LIN {X 152.500,Y 49.993,Z 45.000,A 180.000,B 0.000,C 180.000} C_DIS
LIN {X 152.500,Y 49.993,Z 52.000,A 180.000,B 0.000,C 180.000} C_DIS
LIN {X 147.273,Y 49.993,Z 52.000,A 180.000,B 0.000,C 180.000} C_DIS
LIN {X 147.273,Y 49.993,Z 57.000,A 180.000,B 0.000,C 180.000} C_DIS
LIN {X 118.528,Y 49.993,Z 57.000,A 180.000,B 0.000,C 180.000} C_DIS
LIN {X 118.528,Y 49.993,Z 62.000,A 180.000,B 0.000,C 180.000} C_DIS
LIN {X 104.744,Y 49.993,Z 62.000,A 180.000,B 0.000,C 180.000} C_DIS
LIN {X 104.744,Y 49.993,Z 63.247,A 180.000,B 0.000,C 180.000} C_DIS
LIN {X 104.720,Y 49.993,Z 63.811,A 180.000,B 0.000,C 180.000} C_DIS
LIN {X 104.656,Y 49.993,Z 64.331,A 180.000,B 0.000,C 180.000} C_DIS
LIN {X 104.555,Y 49.993,Z 64.841,A 180.000,B 0.000,C 180.000} C_DIS
LIN {X 104.417,Y 49.993,Z 65.337,A 180.000,B 0.000,C 180.000} C_DIS
LIN {X 104.239,Y 49.993,Z 65.829,A 180.000,B 0.000,C 180.000} C_DIS
LIN {X 104.023,Y 49.993,Z 66.308,A 180.000,B 0.000,C 180.000} C_DIS
LIN {X 103.772,Y 49.993,Z 66.769,A 180.000,B 0.000,C 180.000} C_DIS
LIN {X 103.485,Y 49.993,Z 67.212,A 180.000,B 0.000,C 180.000} C_DIS
LIN {X 103.167,Y 49.993,Z 67.630,A 180.000,B 0.000,C 180.000} C_DIS
LIN {X 102.799,Y 49.993,Z 68.043,A 180.000,B 0.000,C 180.000} C_DIS
LIN {X 102.416,Y 49.993,Z 68.409,A 180.000,B 0.000,C 180.000} C_DIS
LIN {X 102.020,Y 49.993,Z 68.735,A 180.000,B 0.000,C 180.000} C_DIS
LIN {X 101.582,Y 49.993,Z 69.044,A 180.000,B 0.000,C 180.000} C_DIS
LIN {X 101.120,Y 49.993,Z 69.322,A 180.000,B 0.000,C 180.000} C_DIS
LIN {X 100.633,Y 49.993,Z 69.567,A 180.000,B 0.000,C 180.000} C_DIS
LIN {X 100.135,Y 49.993,Z 69.771,A 180.000,B 0.000,C 180.000} C_DIS
LIN {X 99.619,Y 49.993,Z 69.940,A 180.000,B 0.000,C 180.000} C_DIS
LIN {X 99.066,Y 49.993,Z 70.078,A 180.000,B 0.000,C 180.000} C_DIS
LIN {X 98.519,Y 49.993,Z 70.171,A 180.000,B 0.000,C 180.000} C_DIS
LIN {X 97.977,Y 49.993,Z 70.227,A 180.000,B 0.000,C 180.000} C_DIS
LIN {X 97.314,Y 49.993,Z 70.247,A 180.000,B 0.000,C 180.000} C_DIS
LIN {X 95.979,Y 49.993,Z 70.247,A 180.000,B 0.000,C 180.000} C_DIS
LIN {X 95.978,Y 49.993,Z 72.155,A 180.000,B 0.000,C 180.000} C_DIS
LIN {X 90.667,Y 49.993,Z 74.364,A 180.000,B 0.000,C 180.000} C_DIS
LIN {X 85.391,Y 49.993,Z 74.361,A 180.000,B 0.000,C 180.000} C_DIS
LIN {X 84.621,Y 49.993,Z 73.716,A 180.000,B 0.000,C 180.000} C_DIS
LIN {X 83.893,Y 49.993,Z 73.150,A 180.000,B 0.000,C 180.000} C_DIS
LIN {X 83.135,Y 49.993,Z 72.607,A 180.000,B 0.000,C 180.000} C_DIS
LIN {X 82.449,Y 49.993,Z 72.157,A 180.000,B 0.000,C 180.000} C_DIS
LIN {X 81.782,Y 49.993,Z 71.760,A 180.000,B 0.000,C 180.000} C_DIS
LIN {X 81.128,Y 49.993,Z 71.411,A 180.000,B 0.000,C 180.000} C_DIS
LIN {X 80.479,Y 49.993,Z 71.101,A 180.000,B 0.000,C 180.000} C_DIS
LIN {X 79.861,Y 49.993,Z 70.843,A 180.000,B 0.000,C 180.000} C_DIS
LIN {X 79.251,Y 49.993,Z 70.625,A 180.000,B 0.000,C 180.000} C_DIS
LIN {X 78.642,Y 49.993,Z 70.441,A 180.000,B 0.000,C 180.000} C_DIS
LIN {X 78.537,Y 49.993,Z 70.415,A 180.000,B 0.000,C 180.000} C_DIS
LIN {X 78.116,Y 49.993,Z 70.531,A 180.000,B 0.000,C 180.000} C_DIS
LIN {X 77.493,Y 49.993,Z 70.735,A 180.000,B 0.000,C 180.000} C_DIS
LIN {X 76.864,Y 49.993,Z 70.978,A 180.000,B 0.000,C 180.000} C_DIS
LIN {X 76.232,Y 49.993,Z 71.257,A 180.000,B 0.000,C 180.000} C_DIS
LIN {X 75.610,Y 49.993,Z 71.566,A 180.000,B 0.000,C 180.000} C_DIS
LIN {X 74.985,Y 49.993,Z 71.907,A 180.000,B 0.000,C 180.000} C_DIS
LIN {X 74.357,Y 49.993,Z 72.279,A 180.000,B 0.000,C 180.000} C_DIS
LIN {X 73.718,Y 49.993,Z 72.687,A 180.000,B 0.000,C 180.000} C_DIS
LIN {X 73.038,Y 49.993,Z 73.149,A 180.000,B 0.000,C 180.000} C_DIS
LIN {X 72.140,Y 49.993,Z 73.798,A 180.000,B 0.000,C 180.000} C_DIS
LIN {X 71.311,Y 49.993,Z 74.436,A 180.000,B 0.000,C 180.000} C_DIS
LIN {X 70.169,Y 49.993,Z 75.345,A 180.000,B 0.000,C 180.000} C_DIS
LIN {X 66.951,Y 49.993,Z 77.983,A 180.000,B 0.000,C 180.000} C_DIS
LIN {X 65.792,Y 49.993,Z 78.895,A 180.000,B 0.000,C 180.000} C_DIS
LIN {X 65.177,Y 49.993,Z 79.359,A 180.000,B 0.000,C 180.000} C_DIS
LIN {X 64.612,Y 49.993,Z 79.770,A 180.000,B 0.000,C 180.000} C_DIS
LIN {X 64.036,Y 49.993,Z 80.171,A 180.000,B 0.000,C 180.000} C_DIS
LIN {X 63.450,Y 49.993,Z 80.559,A 180.000,B 0.000,C 180.000} C_DIS
LIN {X 62.857,Y 49.993,Z 80.929,A 180.000,B 0.000,C 180.000} C_DIS
LIN {X 62.256,Y 49.993,Z 81.279,A 180.000,B 0.000,C 180.000} C_DIS
LIN {X 61.642,Y 49.993,Z 81.610,A 180.000,B 0.000,C 180.000} C_DIS
LIN {X 61.028,Y 49.993,Z 81.911,A 180.000,B 0.000,C 180.000} C_DIS
LIN {X 60.400,Y 49.993,Z 82.187,A 180.000,B 0.000,C 180.000} C_DIS
LIN {X 59.765,Y 49.993,Z 82.432,A 180.000,B 0.000,C 180.000} C_DIS
LIN {X 59.120,Y 49.993,Z 82.646,A 180.000,B 0.000,C 180.000} C_DIS
LIN {X 58.464,Y 49.993,Z 82.825,A 180.000,B 0.000,C 180.000} C_DIS
LIN {X 57.793,Y 49.993,Z 82.968,A 180.000,B 0.000,C 180.000} C_DIS
LIN {X 57.412,Y 49.993,Z 83.031,A 180.000,B 0.000,C 180.000} C_DIS
LIN {X 57.076,Y 49.993,Z 83.075,A 180.000,B 0.000,C 180.000} C_DIS
LIN {X 56.731,Y 49.993,Z 83.110,A 180.000,B 0.000,C 180.000} C_DIS
LIN {X 56.398,Y 49.993,Z 83.133,A 180.000,B 0.000,C 180.000} C_DIS
LIN {X 56.071,Y 49.993,Z 83.146,A 180.000,B 0.000,C 180.000} C_DIS
LIN {X 55.283,Y 49.993,Z 83.150,A 180.000,B 0.000,C 180.000} C_DIS
LIN {X 50.550,Y 49.993,Z 83.146,A 180.000,B 0.000,C 180.000} C_DIS
LIN {X 50.101,Y 49.993,Z 83.124,A 180.000,B 0.000,C 180.000} C_DIS
LIN {X 49.670,Y 49.993,Z 83.075,A 180.000,B 0.000,C 180.000} C_DIS
LIN {X 49.319,Y 49.993,Z 83.017,A 180.000,B 0.000,C 180.000} C_DIS
LIN {X 48.906,Y 49.993,Z 82.926,A 180.000,B 0.000,C 180.000} C_DIS
LIN {X 48.508,Y 49.993,Z 82.808,A 180.000,B 0.000,C 180.000} C_DIS
LIN {X 48.202,Y 49.993,Z 82.700,A 180.000,B 0.000,C 180.000} C_DIS
LIN {X 47.898,Y 49.993,Z 82.574,A 180.000,B 0.000,C 180.000} C_DIS
LIN {X 47.607,Y 49.993,Z 82.435,A 180.000,B 0.000,C 180.000} C_DIS
LIN {X 47.311,Y 49.993,Z 82.272,A 180.000,B 0.000,C 180.000} C_DIS
LIN {X 46.970,Y 49.993,Z 82.051,A 180.000,B 0.000,C 180.000} C_DIS
LIN {X 46.686,Y 49.993,Z 81.832,A 180.000,B 0.000,C 180.000} C_DIS
LIN {X 46.466,Y 49.993,Z 81.631,A 180.000,B 0.000,C 180.000} C_DIS
LIN {X 46.280,Y 49.993,Z 81.428,A 180.000,B 0.000,C 180.000} C_DIS
LIN {X 46.138,Y 49.993,Z 81.234,A 180.000,B 0.000,C 180.000} C_DIS
LIN {X 46.052,Y 49.993,Z 81.067,A 180.000,B 0.000,C 180.000} C_DIS
LIN {X 46.015,Y 49.993,Z 80.948,A 180.000,B 0.000,C 180.000} C_DIS
LIN {X 46.006,Y 49.993,Z 80.865,A 180.000,B 0.000,C 180.000} C_DIS
LIN {X 46.006,Y 49.993,Z 62.000,A 180.000,B 0.000,C 180.000} C_DIS
LIN {X 36.472,Y 49.993,Z 62.000,A 180.000,B 0.000,C 180.000} C_DIS
LIN {X 36.472,Y 49.993,Z 57.000,A 180.000,B 0.000,C 180.000} C_DIS
LIN {X 7.727,Y 49.993,Z 57.000,A 180.000,B 0.000,C 180.000} C_DIS
LIN {X 7.727,Y 49.993,Z 52.000,A 180.000,B 0.000,C 180.000} C_DIS
LIN {X 2.500,Y 49.993,Z 52.000,A 180.000,B 0.000,C 180.000} C_DIS
LIN {X 2.500,Y 49.993,Z 45.000,A 180.000,B 0.000,C 180.000} C_DIS
LIN {X -0.010,Y 49.993,Z 45.000,A 180.000,B 0.000,C 180.000} C_DIS
; Link Move Starts
LIN {X -0.120,Y 49.993,Z 45.026,A 180.000,B 0.000,C 180.000} C_DIS
LIN {X -0.230,Y 49.993,Z 45.051,A 180.000,B 0.000,C 180.000} C_DIS
LIN {X -0.771,Y 50.305,Z 45.051,A 180.000,B 0.000,C 180.000} C_DIS
LIN {X -0.771,Y 50.930,Z 45.051,A 180.000,B 0.000,C 180.000} C_DIS
LIN {X -0.230,Y 51.243,Z 45.051,A 180.000,B 0.000,C 180.000} C_DIS
LIN {X -0.120,Y 51.243,Z 45.026,A 180.000,B 0.000,C 180.000} C_DIS
LIN {X -0.010,Y 51.243,Z 45.000,A 180.000,B 0.000,C 180.000} C_DIS
; Cutting Move Starts
LIN {X 2.500,Y 51.243,Z 45.000,A 180.000,B 0.000,C 180.000} C_DIS
LIN {X 2.500,Y 51.243,Z 52.000,A 180.000,B 0.000,C 180.000} C_DIS
LIN {X 7.251,Y 51.243,Z 52.000,A 180.000,B 0.000,C 180.000} C_DIS
LIN {X 7.251,Y 51.243,Z 57.000,A 180.000,B 0.000,C 180.000} C_DIS
LIN {X 35.222,Y 51.243,Z 57.000,A 180.000,B 0.000,C 180.000} C_DIS
LIN {X 35.222,Y 51.243,Z 62.000,A 180.000,B 0.000,C 180.000} C_DIS
LIN {X 44.115,Y 51.243,Z 62.000,A 180.000,B 0.000,C 180.000} C_DIS
LIN {X 44.117,Y 51.243,Z 80.467,A 180.000,B 0.000,C 180.000} C_DIS
LIN {X 44.271,Y 51.243,Z 80.606,A 180.000,B 0.000,C 180.000} C_DIS
LIN {X 44.597,Y 51.243,Z 80.888,A 180.000,B 0.000,C 180.000} C_DIS
LIN {X 44.947,Y 51.243,Z 81.164,A 180.000,B 0.000,C 180.000} C_DIS
LIN {X 45.375,Y 51.243,Z 81.471,A 180.000,B 0.000,C 180.000} C_DIS
LIN {X 45.822,Y 51.243,Z 81.755,A 180.000,B 0.000,C 180.000} C_DIS
LIN {X 46.192,Y 51.243,Z 81.966,A 180.000,B 0.000,C 180.000} C_DIS
LIN {X 46.558,Y 51.243,Z 82.155,A 180.000,B 0.000,C 180.000} C_DIS
LIN {X 46.947,Y 51.243,Z 82.336,A 180.000,B 0.000,C 180.000} C_DIS
LIN {X 47.425,Y 51.243,Z 82.530,A 180.000,B 0.000,C 180.000} C_DIS
LIN {X 47.877,Y 51.243,Z 82.685,A 180.000,B 0.000,C 180.000} C_DIS
LIN {X 48.271,Y 51.243,Z 82.801,A 180.000,B 0.000,C 180.000} C_DIS
LIN {X 48.688,Y 51.243,Z 82.904,A 180.000,B 0.000,C 180.000} C_DIS
LIN {X 49.230,Y 51.243,Z 83.010,A 180.000,B 0.000,C 180.000} C_DIS
LIN {X 49.667,Y 51.243,Z 83.072,A 180.000,B 0.000,C 180.000} C_DIS
LIN {X 50.108,Y 51.243,Z 83.116,A 180.000,B 0.000,C 180.000} C_DIS
LIN {X 50.473,Y 51.243,Z 83.138,A 180.000,B 0.000,C 180.000} C_DIS
LIN {X 50.806,Y 51.243,Z 83.148,A 180.000,B 0.000,C 180.000} C_DIS
LIN {X 55.704,Y 51.243,Z 83.150,A 180.000,B 0.000,C 180.000} C_DIS
LIN {X 56.493,Y 51.243,Z 83.146,A 180.000,B 0.000,C 180.000} C_DIS
LIN {X 56.819,Y 51.243,Z 83.133,A 180.000,B 0.000,C 180.000} C_DIS
LIN {X 57.153,Y 51.243,Z 83.110,A 180.000,B 0.000,C 180.000} C_DIS
LIN {X 57.497,Y 51.243,Z 83.075,A 180.000,B 0.000,C 180.000} C_DIS
LIN {X 57.833,Y 51.243,Z 83.031,A 180.000,B 0.000,C 180.000} C_DIS
LIN {X 58.213,Y 51.243,Z 82.968,A 180.000,B 0.000,C 180.000} C_DIS
LIN {X 58.886,Y 51.243,Z 82.825,A 180.000,B 0.000,C 180.000} C_DIS
LIN {X 59.541,Y 51.243,Z 82.646,A 180.000,B 0.000,C 180.000} C_DIS
LIN {X 60.187,Y 51.243,Z 82.432,A 180.000,B 0.000,C 180.000} C_DIS
LIN {X 60.822,Y 51.243,Z 82.187,A 180.000,B 0.000,C 180.000} C_DIS
LIN {X 61.450,Y 51.243,Z 81.911,A 180.000,B 0.000,C 180.000} C_DIS
LIN {X 62.064,Y 51.243,Z 81.610,A 180.000,B 0.000,C 180.000} C_DIS
LIN {X 62.677,Y 51.243,Z 81.279,A 180.000,B 0.000,C 180.000} C_DIS
LIN {X 63.279,Y 51.243,Z 80.929,A 180.000,B 0.000,C 180.000} C_DIS
LIN {X 63.872,Y 51.243,Z 80.559,A 180.000,B 0.000,C 180.000} C_DIS
LIN {X 64.458,Y 51.243,Z 80.171,A 180.000,B 0.000,C 180.000} C_DIS
LIN {X 65.033,Y 51.243,Z 79.770,A 180.000,B 0.000,C 180.000} C_DIS
LIN {X 65.598,Y 51.243,Z 79.359,A 180.000,B 0.000,C 180.000} C_DIS
LIN {X 66.214,Y 51.243,Z 78.896,A 180.000,B 0.000,C 180.000} C_DIS
LIN {X 67.373,Y 51.243,Z 77.983,A 180.000,B 0.000,C 180.000} C_DIS
LIN {X 70.591,Y 51.243,Z 75.345,A 180.000,B 0.000,C 180.000} C_DIS
LIN {X 71.733,Y 51.243,Z 74.436,A 180.000,B 0.000,C 180.000} C_DIS
LIN {X 72.562,Y 51.243,Z 73.798,A 180.000,B 0.000,C 180.000} C_DIS
LIN {X 73.460,Y 51.243,Z 73.149,A 180.000,B 0.000,C 180.000} C_DIS
LIN {X 74.139,Y 51.243,Z 72.687,A 180.000,B 0.000,C 180.000} C_DIS
LIN {X 74.779,Y 51.243,Z 72.279,A 180.000,B 0.000,C 180.000} C_DIS
LIN {X 75.406,Y 51.243,Z 71.907,A 180.000,B 0.000,C 180.000} C_DIS
LIN {X 76.031,Y 51.243,Z 71.566,A 180.000,B 0.000,C 180.000} C_DIS
LIN {X 76.653,Y 51.243,Z 71.257,A 180.000,B 0.000,C 180.000} C_DIS
LIN {X 77.286,Y 51.243,Z 70.978,A 180.000,B 0.000,C 180.000} C_DIS
LIN {X 77.914,Y 51.243,Z 70.735,A 180.000,B 0.000,C 180.000} C_DIS
LIN {X 78.537,Y 51.243,Z 70.531,A 180.000,B 0.000,C 180.000} C_DIS
LIN {X 78.959,Y 51.243,Z 70.415,A 180.000,B 0.000,C 180.000} C_DIS
LIN {X 79.064,Y 51.243,Z 70.441,A 180.000,B 0.000,C 180.000} C_DIS
LIN {X 79.672,Y 51.243,Z 70.625,A 180.000,B 0.000,C 180.000} C_DIS
LIN {X 80.283,Y 51.243,Z 70.843,A 180.000,B 0.000,C 180.000} C_DIS
LIN {X 80.901,Y 51.243,Z 71.101,A 180.000,B 0.000,C 180.000} C_DIS
LIN {X 81.550,Y 51.243,Z 71.411,A 180.000,B 0.000,C 180.000} C_DIS
LIN {X 82.204,Y 51.243,Z 71.760,A 180.000,B 0.000,C 180.000} C_DIS
LIN {X 82.871,Y 51.243,Z 72.157,A 180.000,B 0.000,C 180.000} C_DIS
LIN {X 83.557,Y 51.243,Z 72.607,A 180.000,B 0.000,C 180.000} C_DIS
LIN {X 84.314,Y 51.243,Z 73.150,A 180.000,B 0.000,C 180.000} C_DIS
LIN {X 85.043,Y 51.243,Z 73.716,A 180.000,B 0.000,C 180.000} C_DIS
LIN {X 85.812,Y 51.243,Z 74.361,A 180.000,B 0.000,C 180.000} C_DIS
LIN {X 91.091,Y 51.243,Z 74.364,A 180.000,B 0.000,C 180.000} C_DIS
LIN {X 96.400,Y 51.243,Z 72.155,A 180.000,B 0.000,C 180.000} C_DIS
LIN {X 96.401,Y 51.243,Z 70.247,A 180.000,B 0.000,C 180.000} C_DIS
LIN {X 96.436,Y 51.243,Z 70.247,A 180.000,B 0.000,C 180.000} C_DIS
LIN {X 97.201,Y 51.243,Z 70.228,A 180.000,B 0.000,C 180.000} C_DIS
LIN {X 97.835,Y 51.243,Z 70.171,A 180.000,B 0.000,C 180.000} C_DIS
LIN {X 98.445,Y 51.243,Z 70.077,A 180.000,B 0.000,C 180.000} C_DIS
LIN {X 99.048,Y 51.243,Z 69.941,A 180.000,B 0.000,C 180.000} C_DIS
LIN {X 99.604,Y 51.243,Z 69.772,A 180.000,B 0.000,C 180.000} C_DIS
LIN {X 100.142,Y 51.243,Z 69.564,A 180.000,B 0.000,C 180.000} C_DIS
LIN {X 100.650,Y 51.243,Z 69.326,A 180.000,B 0.000,C 180.000} C_DIS
LIN {X 101.144,Y 51.243,Z 69.043,A 180.000,B 0.000,C 180.000} C_DIS
LIN {X 101.601,Y 51.243,Z 68.735,A 180.000,B 0.000,C 180.000} C_DIS
LIN {X 102.028,Y 51.243,Z 68.398,A 180.000,B 0.000,C 180.000} C_DIS
LIN {X 102.427,Y 51.243,Z 68.030,A 180.000,B 0.000,C 180.000} C_DIS
LIN {X 102.794,Y 51.243,Z 67.630,A 180.000,B 0.000,C 180.000} C_DIS
LIN {X 103.123,Y 51.243,Z 67.212,A 180.000,B 0.000,C 180.000} C_DIS
LIN {X 103.421,Y 51.243,Z 66.768,A 180.000,B 0.000,C 180.000} C_DIS
LIN {X 103.681,Y 51.243,Z 66.307,A 180.000,B 0.000,C 180.000} C_DIS
LIN {X 103.905,Y 51.243,Z 65.828,A 180.000,B 0.000,C 180.000} C_DIS
LIN {X 104.090,Y 51.243,Z 65.333,A 180.000,B 0.000,C 180.000} C_DIS
LIN {X 104.228,Y 51.243,Z 64.853,A 180.000,B 0.000,C 180.000} C_DIS
LIN {X 104.335,Y 51.243,Z 64.336,A 180.000,B 0.000,C 180.000} C_DIS
LIN {X 104.400,Y 51.243,Z 63.822,A 180.000,B 0.000,C 180.000} C_DIS
LIN {X 104.422,Y 51.243,Z 63.353,A 180.000,B 0.000,C 180.000} C_DIS
LIN {X 104.427,Y 51.243,Z 62.000,A 180.000,B 0.000,C 180.000} C_DIS
LIN {X 119.778,Y 51.243,Z 62.000,A 180.000,B 0.000,C 180.000} C_DIS
LIN {X 119.778,Y 51.243,Z 57.000,A 180.000,B 0.000,C 180.000} C_DIS
LIN {X 147.749,Y 51.243,Z 57.000,A 180.000,B 0.000,C 180.000} C_DIS
LIN {X 147.749,Y 51.243,Z 52.000,A 180.000,B 0.000,C 180.000} C_DIS
LIN {X 152.500,Y 51.243,Z 52.000,A 180.000,B 0.000,C 180.000} C_DIS
LIN {X 152.500,Y 51.243,Z 45.000,A 180.000,B 0.000,C 180.000} C_DIS
LIN {X 155.010,Y 51.243,Z 45.000,A 180.000,B 0.000,C 180.000} C_DIS
; Link Move Starts
LIN {X 155.120,Y 51.243,Z 45.026,A 180.000,B 0.000,C 180.000} C_DIS
LIN {X 155.230,Y 51.243,Z 45.051,A 180.000,B 0.000,C 180.000} C_DIS
LIN {X 155.771,Y 51.555,Z 45.051,A 180.000,B 0.000,C 180.000} C_DIS
LIN {X 155.771,Y 52.180,Z 45.051,A 180.000,B 0.000,C 180.000} C_DIS
LIN {X 155.230,Y 52.492,Z 45.051,A 180.000,B 0.000,C 180.000} C_DIS
LIN {X 155.120,Y 52.492,Z 45.026,A 180.000,B 0.000,C 180.000} C_DIS
LIN {X 155.010,Y 52.492,Z 45.000,A 180.000,B 0.000,C 180.000} C_DIS
; Cutting Move Starts
LIN {X 152.500,Y 52.492,Z 45.000,A 180.000,B 0.000,C 180.000} C_DIS
LIN {X 152.500,Y 52.492,Z 52.000,A 180.000,B 0.000,C 180.000} C_DIS
LIN {X 148.203,Y 52.492,Z 52.000,A 180.000,B 0.000,C 180.000} C_DIS
LIN {X 148.199,Y 52.492,Z 57.000,A 180.000,B 0.000,C 180.000} C_DIS
LIN {X 121.028,Y 52.492,Z 57.000,A 180.000,B 0.000,C 180.000} C_DIS
LIN {X 121.028,Y 52.492,Z 62.000,A 180.000,B 0.000,C 180.000} C_DIS
LIN {X 103.956,Y 52.492,Z 62.000,A 180.000,B 0.000,C 180.000} C_DIS
LIN {X 103.953,Y 52.492,Z 63.301,A 180.000,B 0.000,C 180.000} C_DIS
LIN {X 103.931,Y 52.492,Z 63.800,A 180.000,B 0.000,C 180.000} C_DIS
LIN {X 103.865,Y 52.492,Z 64.320,A 180.000,B 0.000,C 180.000} C_DIS
LIN {X 103.757,Y 52.492,Z 64.831,A 180.000,B 0.000,C 180.000} C_DIS
LIN {X 103.610,Y 52.492,Z 65.333,A 180.000,B 0.000,C 180.000} C_DIS
LIN {X 103.411,Y 52.492,Z 65.843,A 180.000,B 0.000,C 180.000} C_DIS
LIN {X 103.185,Y 52.492,Z 66.305,A 180.000,B 0.000,C 180.000} C_DIS
LIN {X 102.912,Y 52.492,Z 66.765,A 180.000,B 0.000,C 180.000} C_DIS
LIN {X 102.599,Y 52.492,Z 67.209,A 180.000,B 0.000,C 180.000} C_DIS
LIN {X 102.251,Y 52.492,Z 67.628,A 180.000,B 0.000,C 180.000} C_DIS
LIN {X 101.862,Y 52.492,Z 68.029,A 180.000,B 0.000,C 180.000} C_DIS
LIN {X 101.440,Y 52.492,Z 68.395,A 180.000,B 0.000,C 180.000} C_DIS
LIN {X 100.981,Y 52.492,Z 68.734,A 180.000,B 0.000,C 180.000} C_DIS
LIN {X 100.490,Y 52.492,Z 69.044,A 180.000,B 0.000,C 180.000} C_DIS
LIN {X 99.962,Y 52.492,Z 69.319,A 180.000,B 0.000,C 180.000} C_DIS
LIN {X 99.400,Y 52.492,Z 69.562,A 180.000,B 0.000,C 180.000} C_DIS
LIN {X 98.791,Y 52.492,Z 69.772,A 180.000,B 0.000,C 180.000} C_DIS
LIN {X 98.157,Y 52.492,Z 69.940,A 180.000,B 0.000,C 180.000} C_DIS
LIN {X 97.461,Y 52.492,Z 70.075,A 180.000,B 0.000,C 180.000} C_DIS
LIN {X 96.823,Y 52.492,Z 70.157,A 180.000,B 0.000,C 180.000} C_DIS
LIN {X 96.820,Y 52.492,Z 72.156,A 180.000,B 0.000,C 180.000} C_DIS
LIN {X 91.513,Y 52.492,Z 74.364,A 180.000,B 0.000,C 180.000} C_DIS
LIN {X 86.234,Y 52.492,Z 74.361,A 180.000,B 0.000,C 180.000} C_DIS
LIN {X 85.465,Y 52.492,Z 73.716,A 180.000,B 0.000,C 180.000} C_DIS
LIN {X 84.737,Y 52.492,Z 73.150,A 180.000,B 0.000,C 180.000} C_DIS
LIN {X 83.979,Y 52.492,Z 72.607,A 180.000,B 0.000,C 180.000} C_DIS
LIN {X 83.293,Y 52.492,Z 72.157,A 180.000,B 0.000,C 180.000} C_DIS
LIN {X 82.626,Y 52.492,Z 71.761,A 180.000,B 0.000,C 180.000} C_DIS
LIN {X 81.972,Y 52.492,Z 71.411,A 180.000,B 0.000,C 180.000} C_DIS
LIN {X 81.323,Y 52.492,Z 71.101,A 180.000,B 0.000,C 180.000} C_DIS
LIN {X 80.705,Y 52.492,Z 70.843,A 180.000,B 0.000,C 180.000} C_DIS
LIN {X 80.085,Y 52.492,Z 70.622,A 180.000,B 0.000,C 180.000} C_DIS
LIN {X 79.463,Y 52.492,Z 70.435,A 180.000,B 0.000,C 180.000} C_DIS
LIN {X 79.381,Y 52.492,Z 70.415,A 180.000,B 0.000,C 180.000} C_DIS
LIN {X 78.959,Y 52.492,Z 70.531,A 180.000,B 0.000,C 180.000} C_DIS
LIN {X 78.336,Y 52.492,Z 70.735,A 180.000,B 0.000,C 180.000} C_DIS
LIN {X 77.707,Y 52.492,Z 70.978,A 180.000,B 0.000,C 180.000} C_DIS
LIN {X 77.075,Y 52.492,Z 71.257,A 180.000,B 0.000,C 180.000} C_DIS
LIN {X 76.453,Y 52.492,Z 71.566,A 180.000,B 0.000,C 180.000} C_DIS
LIN {X 75.828,Y 52.492,Z 71.907,A 180.000,B 0.000,C 180.000} C_DIS
LIN {X 75.200,Y 52.492,Z 72.279,A 180.000,B 0.000,C 180.000} C_DIS
LIN {X 74.561,Y 52.492,Z 72.687,A 180.000,B 0.000,C 180.000} C_DIS
LIN {X 73.881,Y 52.492,Z 73.149,A 180.000,B 0.000,C 180.000} C_DIS
LIN {X 72.984,Y 52.492,Z 73.798,A 180.000,B 0.000,C 180.000} C_DIS
LIN {X 72.154,Y 52.492,Z 74.436,A 180.000,B 0.000,C 180.000} C_DIS
LIN {X 71.013,Y 52.492,Z 75.345,A 180.000,B 0.000,C 180.000} C_DIS
LIN {X 67.794,Y 52.492,Z 77.983,A 180.000,B 0.000,C 180.000} C_DIS
LIN {X 66.636,Y 52.492,Z 78.896,A 180.000,B 0.000,C 180.000} C_DIS
LIN {X 66.020,Y 52.492,Z 79.359,A 180.000,B 0.000,C 180.000} C_DIS
LIN {X 65.455,Y 52.492,Z 79.770,A 180.000,B 0.000,C 180.000} C_DIS
LIN {X 64.879,Y 52.492,Z 80.171,A 180.000,B 0.000,C 180.000} C_DIS
LIN {X 64.294,Y 52.492,Z 80.559,A 180.000,B 0.000,C 180.000} C_DIS
LIN {X 63.700,Y 52.492,Z 80.929,A 180.000,B 0.000,C 180.000} C_DIS
LIN {X 63.099,Y 52.492,Z 81.279,A 180.000,B 0.000,C 180.000} C_DIS
LIN {X 62.485,Y 52.492,Z 81.610,A 180.000,B 0.000,C 180.000} C_DIS
LIN {X 61.872,Y 52.492,Z 81.911,A 180.000,B 0.000,C 180.000} C_DIS
LIN {X 61.243,Y 52.492,Z 82.187,A 180.000,B 0.000,C 180.000} C_DIS
LIN {X 60.608,Y 52.492,Z 82.432,A 180.000,B 0.000,C 180.000} C_DIS
LIN {X 59.963,Y 52.492,Z 82.646,A 180.000,B 0.000,C 180.000} C_DIS
LIN {X 59.308,Y 52.492,Z 82.825,A 180.000,B 0.000,C 180.000} C_DIS
LIN {X 58.634,Y 52.492,Z 82.968,A 180.000,B 0.000,C 180.000} C_DIS
LIN {X 58.255,Y 52.492,Z 83.031,A 180.000,B 0.000,C 180.000} C_DIS
LIN {X 57.919,Y 52.492,Z 83.075,A 180.000,B 0.000,C 180.000} C_DIS
LIN {X 57.570,Y 52.492,Z 83.110,A 180.000,B 0.000,C 180.000} C_DIS
LIN {X 57.241,Y 52.492,Z 83.133,A 180.000,B 0.000,C 180.000} C_DIS
LIN {X 56.914,Y 52.492,Z 83.146,A 180.000,B 0.000,C 180.000} C_DIS
LIN {X 56.125,Y 52.492,Z 83.150,A 180.000,B 0.000,C 180.000} C_DIS
LIN {X 51.228,Y 52.492,Z 83.148,A 180.000,B 0.000,C 180.000} C_DIS
LIN {X 50.894,Y 52.492,Z 83.138,A 180.000,B 0.000,C 180.000} C_DIS
LIN {X 50.551,Y 52.492,Z 83.118,A 180.000,B 0.000,C 180.000} C_DIS
LIN {X 50.192,Y 52.492,Z 83.085,A 180.000,B 0.000,C 180.000} C_DIS
LIN {X 49.834,Y 52.492,Z 83.040,A 180.000,B 0.000,C 180.000} C_DIS
LIN {X 49.459,Y 52.492,Z 82.981,A 180.000,B 0.000,C 180.000} C_DIS
LIN {X 49.097,Y 52.492,Z 82.912,A 180.000,B 0.000,C 180.000} C_DIS
LIN {X 48.722,Y 52.492,Z 82.827,A 180.000,B 0.000,C 180.000} C_DIS
LIN {X 48.335,Y 52.492,Z 82.727,A 180.000,B 0.000,C 180.000} C_DIS
LIN {X 47.958,Y 52.492,Z 82.617,A 180.000,B 0.000,C 180.000} C_DIS
LIN {X 47.571,Y 52.492,Z 82.491,A 180.000,B 0.000,C 180.000} C_DIS
LIN {X 47.180,Y 52.492,Z 82.351,A 180.000,B 0.000,C 180.000} C_DIS
LIN {X 46.794,Y 52.492,Z 82.199,A 180.000,B 0.000,C 180.000} C_DIS
LIN {X 46.392,Y 52.492,Z 82.028,A 180.000,B 0.000,C 180.000} C_DIS
LIN {X 45.925,Y 52.492,Z 81.809,A 180.000,B 0.000,C 180.000} C_DIS
LIN {X 45.499,Y 52.492,Z 81.589,A 180.000,B 0.000,C 180.000} C_DIS
LIN {X 45.076,Y 52.492,Z 81.351,A 180.000,B 0.000,C 180.000} C_DIS
LIN {X 44.646,Y 52.492,Z 81.088,A 180.000,B 0.000,C 180.000} C_DIS
LIN {X 44.123,Y 52.492,Z 80.738,A 180.000,B 0.000,C 180.000} C_DIS
LIN {X 43.749,Y 52.492,Z 80.467,A 180.000,B 0.000,C 180.000} C_DIS
LIN {X 43.747,Y 52.492,Z 62.000,A 180.000,B 0.000,C 180.000} C_DIS
LIN {X 33.972,Y 52.492,Z 62.000,A 180.000,B 0.000,C 180.000} C_DIS
LIN {X 33.972,Y 52.492,Z 57.000,A 180.000,B 0.000,C 180.000} C_DIS
LIN {X 6.797,Y 52.492,Z 57.000,A 180.000,B 0.000,C 180.000} C_DIS
LIN {X 6.797,Y 52.492,Z 52.000,A 180.000,B 0.000,C 180.000} C_DIS
LIN {X 2.500,Y 52.492,Z 52.000,A 180.000,B 0.000,C 180.000} C_DIS
LIN {X 2.500,Y 52.492,Z 45.000,A 180.000,B 0.000,C 180.000} C_DIS
LIN {X -0.010,Y 52.492,Z 45.000,A 180.000,B 0.000,C 180.000} C_DIS
; Link Move Starts
LIN {X -0.120,Y 52.492,Z 45.026,A 180.000,B 0.000,C 180.000} C_DIS
LIN {X -0.230,Y 52.492,Z 45.051,A 180.000,B 0.000,C 180.000} C_DIS
LIN {X -0.771,Y 52.805,Z 45.051,A 180.000,B 0.000,C 180.000} C_DIS
LIN {X -0.771,Y 53.430,Z 45.051,A 180.000,B 0.000,C 180.000} C_DIS
LIN {X -0.230,Y 53.742,Z 45.051,A 180.000,B 0.000,C 180.000} C_DIS
LIN {X -0.120,Y 53.742,Z 45.026,A 180.000,B 0.000,C 180.000} C_DIS
LIN {X -0.010,Y 53.742,Z 45.000,A 180.000,B 0.000,C 180.000} C_DIS
; Cutting Move Starts
LIN {X 2.500,Y 53.742,Z 45.000,A 180.000,B 0.000,C 180.000} C_DIS
LIN {X 2.500,Y 53.742,Z 52.000,A 180.000,B 0.000,C 180.000} C_DIS
LIN {X 6.366,Y 53.742,Z 52.000,A 180.000,B 0.000,C 180.000} C_DIS
LIN {X 6.366,Y 53.742,Z 57.000,A 180.000,B 0.000,C 180.000} C_DIS
LIN {X 32.717,Y 53.742,Z 57.000,A 180.000,B 0.000,C 180.000} C_DIS
LIN {X 32.722,Y 53.742,Z 62.000,A 180.000,B 0.000,C 180.000} C_DIS
LIN {X 44.012,Y 53.742,Z 62.000,A 180.000,B 0.000,C 180.000} C_DIS
LIN {X 44.012,Y 53.742,Z 80.467,A 180.000,B 0.000,C 180.000} C_DIS
LIN {X 44.345,Y 53.742,Z 80.684,A 180.000,B 0.000,C 180.000} C_DIS
LIN {X 44.765,Y 53.742,Z 80.947,A 180.000,B 0.000,C 180.000} C_DIS
LIN {X 45.184,Y 53.742,Z 81.196,A 180.000,B 0.000,C 180.000} C_DIS
LIN {X 45.599,Y 53.742,Z 81.428,A 180.000,B 0.000,C 180.000} C_DIS
LIN {X 46.008,Y 53.742,Z 81.643,A 180.000,B 0.000,C 180.000} C_DIS
LIN {X 46.412,Y 53.742,Z 81.843,A 180.000,B 0.000,C 180.000} C_DIS
LIN {X 46.812,Y 53.742,Z 82.027,A 180.000,B 0.000,C 180.000} C_DIS
LIN {X 47.209,Y 53.742,Z 82.196,A 180.000,B 0.000,C 180.000} C_DIS
LIN {X 47.602,Y 53.742,Z 82.351,A 180.000,B 0.000,C 180.000} C_DIS
LIN {X 47.992,Y 53.742,Z 82.491,A 180.000,B 0.000,C 180.000} C_DIS
LIN {X 48.380,Y 53.742,Z 82.617,A 180.000,B 0.000,C 180.000} C_DIS
LIN {X 48.757,Y 53.742,Z 82.727,A 180.000,B 0.000,C 180.000} C_DIS
LIN {X 49.144,Y 53.742,Z 82.827,A 180.000,B 0.000,C 180.000} C_DIS
LIN {X 49.519,Y 53.742,Z 82.912,A 180.000,B 0.000,C 180.000} C_DIS
LIN {X 49.880,Y 53.742,Z 82.981,A 180.000,B 0.000,C 180.000} C_DIS
LIN {X 50.256,Y 53.742,Z 83.040,A 180.000,B 0.000,C 180.000} C_DIS
LIN {X 50.613,Y 53.742,Z 83.085,A 180.000,B 0.000,C 180.000} C_DIS
LIN {X 50.969,Y 53.742,Z 83.117,A 180.000,B 0.000,C 180.000} C_DIS
LIN {X 51.316,Y 53.742,Z 83.138,A 180.000,B 0.000,C 180.000} C_DIS
LIN {X 51.650,Y 53.742,Z 83.148,A 180.000,B 0.000,C 180.000} C_DIS
LIN {X 56.547,Y 53.742,Z 83.150,A 180.000,B 0.000,C 180.000} C_DIS
LIN {X 57.336,Y 53.742,Z 83.146,A 180.000,B 0.000,C 180.000} C_DIS
LIN {X 57.663,Y 53.742,Z 83.133,A 180.000,B 0.000,C 180.000} C_DIS
LIN {X 57.992,Y 53.742,Z 83.110,A 180.000,B 0.000,C 180.000} C_DIS
LIN {X 58.341,Y 53.742,Z 83.075,A 180.000,B 0.000,C 180.000} C_DIS
LIN {X 58.677,Y 53.742,Z 83.031,A 180.000,B 0.000,C 180.000} C_DIS
LIN {X 59.056,Y 53.742,Z 82.968,A 180.000,B 0.000,C 180.000} C_DIS
LIN {X 59.729,Y 53.742,Z 82.825,A 180.000,B 0.000,C 180.000} C_DIS
LIN {X 60.385,Y 53.742,Z 82.646,A 180.000,B 0.000,C 180.000} C_DIS
LIN {X 61.030,Y 53.742,Z 82.432,A 180.000,B 0.000,C 180.000} C_DIS
LIN {X 61.665,Y 53.742,Z 82.187,A 180.000,B 0.000,C 180.000} C_DIS
LIN {X 62.293,Y 53.742,Z 81.911,A 180.000,B 0.000,C 180.000} C_DIS
LIN {X 62.907,Y 53.742,Z 81.610,A 180.000,B 0.000,C 180.000} C_DIS
LIN {X 63.521,Y 53.742,Z 81.279,A 180.000,B 0.000,C 180.000} C_DIS
LIN {X 64.122,Y 53.742,Z 80.929,A 180.000,B 0.000,C 180.000} C_DIS
LIN {X 64.715,Y 53.742,Z 80.559,A 180.000,B 0.000,C 180.000} C_DIS
LIN {X 65.301,Y 53.742,Z 80.171,A 180.000,B 0.000,C 180.000} C_DIS
LIN {X 65.877,Y 53.742,Z 79.770,A 180.000,B 0.000,C 180.000} C_DIS
LIN {X 66.442,Y 53.742,Z 79.359,A 180.000,B 0.000,C 180.000} C_DIS
LIN {X 67.057,Y 53.742,Z 78.895,A 180.000,B 0.000,C 180.000} C_DIS
LIN {X 68.216,Y 53.742,Z 77.983,A 180.000,B 0.000,C 180.000} C_DIS
LIN {X 71.434,Y 53.742,Z 75.345,A 180.000,B 0.000,C 180.000} C_DIS
LIN {X 72.576,Y 53.742,Z 74.436,A 180.000,B 0.000,C 180.000} C_DIS
LIN {X 73.405,Y 53.742,Z 73.798,A 180.000,B 0.000,C 180.000} C_DIS
LIN {X 74.303,Y 53.742,Z 73.149,A 180.000,B 0.000,C 180.000} C_DIS
LIN {X 74.983,Y 53.742,Z 72.687,A 180.000,B 0.000,C 180.000} C_DIS
LIN {X 75.622,Y 53.742,Z 72.279,A 180.000,B 0.000,C 180.000} C_DIS
LIN {X 76.250,Y 53.742,Z 71.907,A 180.000,B 0.000,C 180.000} C_DIS
LIN {X 76.875,Y 53.742,Z 71.566,A 180.000,B 0.000,C 180.000} C_DIS
LIN {X 77.497,Y 53.742,Z 71.257,A 180.000,B 0.000,C 180.000} C_DIS
LIN {X 78.129,Y 53.742,Z 70.978,A 180.000,B 0.000,C 180.000} C_DIS
LIN {X 78.758,Y 53.742,Z 70.735,A 180.000,B 0.000,C 180.000} C_DIS
LIN {X 79.381,Y 53.742,Z 70.531,A 180.000,B 0.000,C 180.000} C_DIS
LIN {X 79.803,Y 53.742,Z 70.415,A 180.000,B 0.000,C 180.000} C_DIS
LIN {X 79.885,Y 53.742,Z 70.435,A 180.000,B 0.000,C 180.000} C_DIS
LIN {X 80.508,Y 53.742,Z 70.622,A 180.000,B 0.000,C 180.000} C_DIS
LIN {X 81.128,Y 53.742,Z 70.844,A 180.000,B 0.000,C 180.000} C_DIS
LIN {X 81.746,Y 53.742,Z 71.102,A 180.000,B 0.000,C 180.000} C_DIS
LIN {X 82.394,Y 53.742,Z 71.411,A 180.000,B 0.000,C 180.000} C_DIS
LIN {X 83.048,Y 53.742,Z 71.761,A 180.000,B 0.000,C 180.000} C_DIS
LIN {X 83.715,Y 53.742,Z 72.158,A 180.000,B 0.000,C 180.000} C_DIS
LIN {X 84.401,Y 53.742,Z 72.608,A 180.000,B 0.000,C 180.000} C_DIS
LIN {X 85.159,Y 53.742,Z 73.150,A 180.000,B 0.000,C 180.000} C_DIS
LIN {X 85.887,Y 53.742,Z 73.717,A 180.000,B 0.000,C 180.000} C_DIS
LIN {X 86.659,Y 53.742,Z 74.364,A 180.000,B 0.000,C 180.000} C_DIS
LIN {X 91.933,Y 53.742,Z 74.364,A 180.000,B 0.000,C 180.000} C_DIS
LIN {X 97.243,Y 53.742,Z 72.156,A 180.000,B 0.000,C 180.000} C_DIS
LIN {X 97.244,Y 53.742,Z 69.838,A 180.000,B 0.000,C 180.000} C_DIS
LIN {X 97.601,Y 53.742,Z 69.760,A 180.000,B 0.000,C 180.000} C_DIS
LIN {X 98.252,Y 53.742,Z 69.574,A 180.000,B 0.000,C 180.000} C_DIS
LIN {X 98.394,Y 53.742,Z 69.527,A 180.000,B 0.000,C 180.000} C_DIS
LIN {X 99.002,Y 53.742,Z 69.299,A 180.000,B 0.000,C 180.000} C_DIS
LIN {X 99.556,Y 53.742,Z 69.043,A 180.000,B 0.000,C 180.000} C_DIS
LIN {X 100.127,Y 53.742,Z 68.725,A 180.000,B 0.000,C 180.000} C_DIS
LIN {X 100.617,Y 53.742,Z 68.393,A 180.000,B 0.000,C 180.000} C_DIS
LIN {X 101.095,Y 53.742,Z 68.014,A 180.000,B 0.000,C 180.000} C_DIS
LIN {X 101.502,Y 53.742,Z 67.630,A 180.000,B 0.000,C 180.000} C_DIS
LIN {X 101.880,Y 53.742,Z 67.207,A 180.000,B 0.000,C 180.000} C_DIS
LIN {X 102.215,Y 53.742,Z 66.764,A 180.000,B 0.000,C 180.000} C_DIS
LIN {X 102.500,Y 53.742,Z 66.319,A 180.000,B 0.000,C 180.000} C_DIS
LIN {X 102.756,Y 53.742,Z 65.823,A 180.000,B 0.000,C 180.000} C_DIS
LIN {X 102.956,Y 53.742,Z 65.333,A 180.000,B 0.000,C 180.000} C_DIS
LIN {X 103.116,Y 53.742,Z 64.822,A 180.000,B 0.000,C 180.000} C_DIS
LIN {X 103.225,Y 53.742,Z 64.328,A 180.000,B 0.000,C 180.000} C_DIS
LIN {X 103.296,Y 53.742,Z 63.810,A 180.000,B 0.000,C 180.000} C_DIS
LIN {X 103.321,Y 53.742,Z 63.314,A 180.000,B 0.000,C 180.000} C_DIS
LIN {X 103.324,Y 53.742,Z 62.000,A 180.000,B 0.000,C 180.000} C_DIS
LIN {X 122.278,Y 53.742,Z 62.000,A 180.000,B 0.000,C 180.000} C_DIS
LIN {X 122.278,Y 53.742,Z 57.000,A 180.000,B 0.000,C 180.000} C_DIS
LIN {X 148.634,Y 53.742,Z 57.000,A 180.000,B 0.000,C 180.000} C_DIS
LIN {X 148.634,Y 53.742,Z 52.000,A 180.000,B 0.000,C 180.000} C_DIS
LIN {X 152.500,Y 53.742,Z 52.000,A 180.000,B 0.000,C 180.000} C_DIS
LIN {X 152.500,Y 53.742,Z 45.000,A 180.000,B 0.000,C 180.000} C_DIS
LIN {X 155.010,Y 53.742,Z 45.000,A 180.000,B 0.000,C 180.000} C_DIS
; Link Move Starts
LIN {X 155.120,Y 53.742,Z 45.026,A 180.000,B 0.000,C 180.000} C_DIS
LIN {X 155.230,Y 53.742,Z 45.051,A 180.000,B 0.000,C 180.000} C_DIS
LIN {X 155.771,Y 54.055,Z 45.051,A 180.000,B 0.000,C 180.000} C_DIS
LIN {X 155.771,Y 54.680,Z 45.051,A 180.000,B 0.000,C 180.000} C_DIS
LIN {X 155.230,Y 54.992,Z 45.051,A 180.000,B 0.000,C 180.000} C_DIS
LIN {X 155.120,Y 54.992,Z 45.026,A 180.000,B 0.000,C 180.000} C_DIS
LIN {X 155.010,Y 54.992,Z 45.000,A 180.000,B 0.000,C 180.000} C_DIS
; Cutting Move Starts
LIN {X 152.500,Y 54.992,Z 45.000,A 180.000,B 0.000,C 180.000} C_DIS
LIN {X 152.500,Y 54.992,Z 52.000,A 180.000,B 0.000,C 180.000} C_DIS
LIN {X 149.043,Y 54.992,Z 52.000,A 180.000,B 0.000,C 180.000} C_DIS
LIN {X 149.041,Y 54.992,Z 57.000,A 180.000,B 0.000,C 180.000} C_DIS
LIN {X 123.528,Y 54.992,Z 57.000,A 180.000,B 0.000,C 180.000} C_DIS
LIN {X 123.528,Y 54.992,Z 62.000,A 180.000,B 0.000,C 180.000} C_DIS
LIN {X 102.500,Y 54.992,Z 62.000,A 180.000,B 0.000,C 180.000} C_DIS
LIN {X 102.497,Y 54.992,Z 63.302,A 180.000,B 0.000,C 180.000} C_DIS
LIN {X 102.470,Y 54.992,Z 63.804,A 180.000,B 0.000,C 180.000} C_DIS
LIN {X 102.393,Y 54.992,Z 64.325,A 180.000,B 0.000,C 180.000} C_DIS
LIN {X 102.268,Y 54.992,Z 64.838,A 180.000,B 0.000,C 180.000} C_DIS
LIN {X 102.103,Y 54.992,Z 65.325,A 180.000,B 0.000,C 180.000} C_DIS
LIN {X 101.881,Y 54.992,Z 65.826,A 180.000,B 0.000,C 180.000} C_DIS
LIN {X 101.614,Y 54.992,Z 66.297,A 180.000,B 0.000,C 180.000} C_DIS
LIN {X 101.288,Y 54.992,Z 66.762,A 180.000,B 0.000,C 180.000} C_DIS
LIN {X 100.916,Y 54.992,Z 67.207,A 180.000,B 0.000,C 180.000} C_DIS
LIN {X 100.518,Y 54.992,Z 67.608,A 180.000,B 0.000,C 180.000} C_DIS
LIN {X 100.015,Y 54.992,Z 68.024,A 180.000,B 0.000,C 180.000} C_DIS
LIN {X 99.581,Y 54.992,Z 68.329,A 180.000,B 0.000,C 180.000} C_DIS
LIN {X 99.466,Y 54.992,Z 68.402,A 180.000,B 0.000,C 180.000} C_DIS
LIN {X 98.889,Y 54.992,Z 68.732,A 180.000,B 0.000,C 180.000} C_DIS
LIN {X 98.217,Y 54.992,Z 69.041,A 180.000,B 0.000,C 180.000} C_DIS
LIN {X 97.741,Y 54.992,Z 69.217,A 180.000,B 0.000,C 180.000} C_DIS
LIN {X 97.666,Y 54.992,Z 69.244,A 180.000,B 0.000,C 180.000} C_DIS
LIN {X 97.664,Y 54.992,Z 72.156,A 180.000,B 0.000,C 180.000} C_DIS
LIN {X 92.353,Y 54.992,Z 74.364,A 180.000,B 0.000,C 180.000} C_DIS
LIN {X 87.081,Y 54.992,Z 74.364,A 180.000,B 0.000,C 180.000} C_DIS
LIN {X 86.309,Y 54.992,Z 73.717,A 180.000,B 0.000,C 180.000} C_DIS
LIN {X 85.581,Y 54.992,Z 73.150,A 180.000,B 0.000,C 180.000} C_DIS
LIN {X 84.823,Y 54.992,Z 72.608,A 180.000,B 0.000,C 180.000} C_DIS
LIN {X 84.137,Y 54.992,Z 72.158,A 180.000,B 0.000,C 180.000} C_DIS
LIN {X 83.470,Y 54.992,Z 71.761,A 180.000,B 0.000,C 180.000} C_DIS
LIN {X 82.816,Y 54.992,Z 71.411,A 180.000,B 0.000,C 180.000} C_DIS
LIN {X 82.167,Y 54.992,Z 71.102,A 180.000,B 0.000,C 180.000} C_DIS
LIN {X 81.549,Y 54.992,Z 70.844,A 180.000,B 0.000,C 180.000} C_DIS
LIN {X 80.930,Y 54.992,Z 70.622,A 180.000,B 0.000,C 180.000} C_DIS
LIN {X 80.307,Y 54.992,Z 70.435,A 180.000,B 0.000,C 180.000} C_DIS
LIN {X 80.225,Y 54.992,Z 70.415,A 180.000,B 0.000,C 180.000} C_DIS
LIN {X 79.803,Y 54.992,Z 70.531,A 180.000,B 0.000,C 180.000} C_DIS
LIN {X 79.179,Y 54.992,Z 70.735,A 180.000,B 0.000,C 180.000} C_DIS
LIN {X 78.551,Y 54.992,Z 70.978,A 180.000,B 0.000,C 180.000} C_DIS
LIN {X 77.918,Y 54.992,Z 71.257,A 180.000,B 0.000,C 180.000} C_DIS
LIN {X 77.296,Y 54.992,Z 71.566,A 180.000,B 0.000,C 180.000} C_DIS
LIN {X 76.671,Y 54.992,Z 71.907,A 180.000,B 0.000,C 180.000} C_DIS
LIN {X 76.044,Y 54.992,Z 72.279,A 180.000,B 0.000,C 180.000} C_DIS
LIN {X 75.404,Y 54.992,Z 72.687,A 180.000,B 0.000,C 180.000} C_DIS
LIN {X 74.725,Y 54.992,Z 73.149,A 180.000,B 0.000,C 180.000} C_DIS
LIN {X 73.827,Y 54.992,Z 73.798,A 180.000,B 0.000,C 180.000} C_DIS
LIN {X 72.998,Y 54.992,Z 74.436,A 180.000,B 0.000,C 180.000} C_DIS
LIN {X 71.856,Y 54.992,Z 75.345,A 180.000,B 0.000,C 180.000} C_DIS
LIN {X 68.638,Y 54.992,Z 77.983,A 180.000,B 0.000,C 180.000} C_DIS
LIN {X 67.479,Y 54.992,Z 78.895,A 180.000,B 0.000,C 180.000} C_DIS
LIN {X 66.863,Y 54.992,Z 79.359,A 180.000,B 0.000,C 180.000} C_DIS
LIN {X 66.298,Y 54.992,Z 79.770,A 180.000,B 0.000,C 180.000} C_DIS
LIN {X 65.723,Y 54.992,Z 80.171,A 180.000,B 0.000,C 180.000} C_DIS
LIN {X 65.137,Y 54.992,Z 80.559,A 180.000,B 0.000,C 180.000} C_DIS
LIN {X 64.544,Y 54.992,Z 80.929,A 180.000,B 0.000,C 180.000} C_DIS
LIN {X 63.943,Y 54.992,Z 81.279,A 180.000,B 0.000,C 180.000} C_DIS
LIN {X 63.329,Y 54.992,Z 81.610,A 180.000,B 0.000,C 180.000} C_DIS
LIN {X 62.715,Y 54.992,Z 81.911,A 180.000,B 0.000,C 180.000} C_DIS
LIN {X 62.087,Y 54.992,Z 82.187,A 180.000,B 0.000,C 180.000} C_DIS
LIN {X 61.452,Y 54.992,Z 82.432,A 180.000,B 0.000,C 180.000} C_DIS
LIN {X 60.807,Y 54.992,Z 82.646,A 180.000,B 0.000,C 180.000} C_DIS
LIN {X 60.151,Y 54.992,Z 82.825,A 180.000,B 0.000,C 180.000} C_DIS
LIN {X 59.478,Y 54.992,Z 82.968,A 180.000,B 0.000,C 180.000} C_DIS
LIN {X 59.098,Y 54.992,Z 83.031,A 180.000,B 0.000,C 180.000} C_DIS
LIN {X 58.762,Y 54.992,Z 83.075,A 180.000,B 0.000,C 180.000} C_DIS
LIN {X 58.414,Y 54.992,Z 83.110,A 180.000,B 0.000,C 180.000} C_DIS
LIN {X 58.084,Y 54.992,Z 83.133,A 180.000,B 0.000,C 180.000} C_DIS
LIN {X 57.758,Y 54.992,Z 83.146,A 180.000,B 0.000,C 180.000} C_DIS
LIN {X 56.969,Y 54.992,Z 83.150,A 180.000,B 0.000,C 180.000} C_DIS
LIN {X 52.071,Y 54.992,Z 83.148,A 180.000,B 0.000,C 180.000} C_DIS
LIN {X 51.737,Y 54.992,Z 83.138,A 180.000,B 0.000,C 180.000} C_DIS
LIN {X 51.391,Y 54.992,Z 83.117,A 180.000,B 0.000,C 180.000} C_DIS
LIN {X 51.035,Y 54.992,Z 83.085,A 180.000,B 0.000,C 180.000} C_DIS
LIN {X 50.678,Y 54.992,Z 83.040,A 180.000,B 0.000,C 180.000} C_DIS
LIN {X 50.300,Y 54.992,Z 82.980,A 180.000,B 0.000,C 180.000} C_DIS
LIN {X 49.941,Y 54.992,Z 82.912,A 180.000,B 0.000,C 180.000} C_DIS
LIN {X 49.564,Y 54.992,Z 82.827,A 180.000,B 0.000,C 180.000} C_DIS
LIN {X 49.178,Y 54.992,Z 82.727,A 180.000,B 0.000,C 180.000} C_DIS
LIN {X 48.802,Y 54.992,Z 82.617,A 180.000,B 0.000,C 180.000} C_DIS
LIN {X 48.414,Y 54.992,Z 82.491,A 180.000,B 0.000,C 180.000} C_DIS
LIN {X 48.023,Y 54.992,Z 82.351,A 180.000,B 0.000,C 180.000} C_DIS
LIN {X 47.630,Y 54.992,Z 82.196,A 180.000,B 0.000,C 180.000} C_DIS
LIN {X 47.234,Y 54.992,Z 82.027,A 180.000,B 0.000,C 180.000} C_DIS
LIN {X 46.833,Y 54.992,Z 81.843,A 180.000,B 0.000,C 180.000} C_DIS
LIN {X 46.429,Y 54.992,Z 81.643,A 180.000,B 0.000,C 180.000} C_DIS
LIN {X 46.020,Y 54.992,Z 81.428,A 180.000,B 0.000,C 180.000} C_DIS
LIN {X 45.606,Y 54.992,Z 81.196,A 180.000,B 0.000,C 180.000} C_DIS
LIN {X 45.186,Y 54.992,Z 80.947,A 180.000,B 0.000,C 180.000} C_DIS
LIN {X 44.766,Y 54.992,Z 80.684,A 180.000,B 0.000,C 180.000} C_DIS
LIN {X 44.434,Y 54.992,Z 80.467,A 180.000,B 0.000,C 180.000} C_DIS
LIN {X 44.434,Y 54.992,Z 62.000,A 180.000,B 0.000,C 180.000} C_DIS
LIN {X 31.472,Y 54.992,Z 62.000,A 180.000,B 0.000,C 180.000} C_DIS
LIN {X 31.471,Y 54.992,Z 57.000,A 180.000,B 0.000,C 180.000} C_DIS
LIN {X 5.957,Y 54.992,Z 57.000,A 180.000,B 0.000,C 180.000} C_DIS
LIN {X 5.957,Y 54.992,Z 52.000,A 180.000,B 0.000,C 180.000} C_DIS
LIN {X 2.500,Y 54.992,Z 52.000,A 180.000,B 0.000,C 180.000} C_DIS
LIN {X 2.498,Y 54.992,Z 45.000,A 180.000,B 0.000,C 180.000} C_DIS
LIN {X -0.010,Y 54.992,Z 45.000,A 180.000,B 0.000,C 180.000} C_DIS
; Link Move Starts
LIN {X -0.120,Y 54.992,Z 45.026,A 180.000,B 0.000,C 180.000} C_DIS
LIN {X -0.230,Y 54.992,Z 45.051,A 180.000,B 0.000,C 180.000} C_DIS
LIN {X -0.771,Y 55.305,Z 45.051,A 180.000,B 0.000,C 180.000} C_DIS
LIN {X -0.771,Y 55.930,Z 45.051,A 180.000,B 0.000,C 180.000} C_DIS
LIN {X -0.230,Y 56.242,Z 45.051,A 180.000,B 0.000,C 180.000} C_DIS
LIN {X -0.120,Y 56.242,Z 45.026,A 180.000,B 0.000,C 180.000} C_DIS
LIN {X -0.010,Y 56.242,Z 45.000,A 180.000,B 0.000,C 180.000} C_DIS
; Cutting Move Starts
LIN {X 2.500,Y 56.242,Z 45.000,A 180.000,B 0.000,C 180.000} C_DIS
LIN {X 2.500,Y 56.242,Z 52.000,A 180.000,B 0.000,C 180.000} C_DIS
LIN {X 5.580,Y 56.242,Z 52.000,A 180.000,B 0.000,C 180.000} C_DIS
LIN {X 5.580,Y 56.242,Z 57.000,A 180.000,B 0.000,C 180.000} C_DIS
LIN {X 30.222,Y 56.242,Z 57.000,A 180.000,B 0.000,C 180.000} C_DIS
LIN {X 30.222,Y 56.242,Z 62.000,A 180.000,B 0.000,C 180.000} C_DIS
LIN {X 44.856,Y 56.242,Z 62.000,A 180.000,B 0.000,C 180.000} C_DIS
LIN {X 44.856,Y 56.242,Z 80.467,A 180.000,B 0.000,C 180.000} C_DIS
LIN {X 45.188,Y 56.242,Z 80.684,A 180.000,B 0.000,C 180.000} C_DIS
LIN {X 45.608,Y 56.242,Z 80.947,A 180.000,B 0.000,C 180.000} C_DIS
LIN {X 46.027,Y 56.242,Z 81.196,A 180.000,B 0.000,C 180.000} C_DIS
LIN {X 46.442,Y 56.242,Z 81.428,A 180.000,B 0.000,C 180.000} C_DIS
LIN {X 46.851,Y 56.242,Z 81.643,A 180.000,B 0.000,C 180.000} C_DIS
LIN {X 47.255,Y 56.242,Z 81.843,A 180.000,B 0.000,C 180.000} C_DIS
LIN {X 47.662,Y 56.242,Z 82.030,A 180.000,B 0.000,C 180.000} C_DIS
LIN {X 48.059,Y 56.242,Z 82.199,A 180.000,B 0.000,C 180.000} C_DIS
LIN {X 48.445,Y 56.242,Z 82.351,A 180.000,B 0.000,C 180.000} C_DIS
LIN {X 48.835,Y 56.242,Z 82.491,A 180.000,B 0.000,C 180.000} C_DIS
LIN {X 49.223,Y 56.242,Z 82.617,A 180.000,B 0.000,C 180.000} C_DIS
LIN {X 49.600,Y 56.242,Z 82.727,A 180.000,B 0.000,C 180.000} C_DIS
LIN {X 49.986,Y 56.242,Z 82.827,A 180.000,B 0.000,C 180.000} C_DIS
LIN {X 50.362,Y 56.242,Z 82.912,A 180.000,B 0.000,C 180.000} C_DIS
LIN {X 50.722,Y 56.242,Z 82.980,A 180.000,B 0.000,C 180.000} C_DIS
LIN {X 51.099,Y 56.242,Z 83.040,A 180.000,B 0.000,C 180.000} C_DIS
LIN {X 51.457,Y 56.242,Z 83.085,A 180.000,B 0.000,C 180.000} C_DIS
LIN {X 51.812,Y 56.242,Z 83.117,A 180.000,B 0.000,C 180.000} C_DIS
LIN {X 52.159,Y 56.242,Z 83.138,A 180.000,B 0.000,C 180.000} C_DIS
LIN {X 52.493,Y 56.242,Z 83.148,A 180.000,B 0.000,C 180.000} C_DIS
LIN {X 57.390,Y 56.242,Z 83.150,A 180.000,B 0.000,C 180.000} C_DIS
LIN {X 58.179,Y 56.242,Z 83.146,A 180.000,B 0.000,C 180.000} C_DIS
LIN {X 58.506,Y 56.242,Z 83.133,A 180.000,B 0.000,C 180.000} C_DIS
LIN {X 58.835,Y 56.242,Z 83.110,A 180.000,B 0.000,C 180.000} C_DIS
LIN {X 59.184,Y 56.242,Z 83.075,A 180.000,B 0.000,C 180.000} C_DIS
LIN {X 59.520,Y 56.242,Z 83.031,A 180.000,B 0.000,C 180.000} C_DIS
LIN {X 59.899,Y 56.242,Z 82.968,A 180.000,B 0.000,C 180.000} C_DIS
LIN {X 60.573,Y 56.242,Z 82.825,A 180.000,B 0.000,C 180.000} C_DIS
LIN {X 61.228,Y 56.242,Z 82.646,A 180.000,B 0.000,C 180.000} C_DIS
LIN {X 61.873,Y 56.242,Z 82.432,A 180.000,B 0.000,C 180.000} C_DIS
LIN {X 62.508,Y 56.242,Z 82.187,A 180.000,B 0.000,C 180.000} C_DIS
LIN {X 63.136,Y 56.242,Z 81.911,A 180.000,B 0.000,C 180.000} C_DIS
LIN {X 63.750,Y 56.242,Z 81.610,A 180.000,B 0.000,C 180.000} C_DIS
LIN {X 64.364,Y 56.242,Z 81.279,A 180.000,B 0.000,C 180.000} C_DIS
LIN {X 64.965,Y 56.242,Z 80.929,A 180.000,B 0.000,C 180.000} C_DIS
LIN {X 65.559,Y 56.242,Z 80.559,A 180.000,B 0.000,C 180.000} C_DIS
LIN {X 66.144,Y 56.242,Z 80.171,A 180.000,B 0.000,C 180.000} C_DIS
LIN {X 66.720,Y 56.242,Z 79.770,A 180.000,B 0.000,C 180.000} C_DIS
LIN {X 67.285,Y 56.242,Z 79.359,A 180.000,B 0.000,C 180.000} C_DIS
LIN {X 67.901,Y 56.242,Z 78.896,A 180.000,B 0.000,C 180.000} C_DIS
LIN {X 69.059,Y 56.242,Z 77.983,A 180.000,B 0.000,C 180.000} C_DIS
LIN {X 72.278,Y 56.242,Z 75.345,A 180.000,B 0.000,C 180.000} C_DIS
LIN {X 73.419,Y 56.242,Z 74.436,A 180.000,B 0.000,C 180.000} C_DIS
LIN {X 74.249,Y 56.242,Z 73.798,A 180.000,B 0.000,C 180.000} C_DIS
LIN {X 75.146,Y 56.242,Z 73.149,A 180.000,B 0.000,C 180.000} C_DIS
LIN {X 75.826,Y 56.242,Z 72.687,A 180.000,B 0.000,C 180.000} C_DIS
LIN {X 76.465,Y 56.242,Z 72.279,A 180.000,B 0.000,C 180.000} C_DIS
LIN {X 77.093,Y 56.242,Z 71.907,A 180.000,B 0.000,C 180.000} C_DIS
LIN {X 77.718,Y 56.242,Z 71.566,A 180.000,B 0.000,C 180.000} C_DIS
LIN {X 78.340,Y 56.242,Z 71.257,A 180.000,B 0.000,C 180.000} C_DIS
LIN {X 78.972,Y 56.242,Z 70.978,A 180.000,B 0.000,C 180.000} C_DIS
LIN {X 79.601,Y 56.242,Z 70.735,A 180.000,B 0.000,C 180.000} C_DIS
LIN {X 80.224,Y 56.242,Z 70.531,A 180.000,B 0.000,C 180.000} C_DIS
LIN {X 80.645,Y 56.242,Z 70.415,A 180.000,B 0.000,C 180.000} C_DIS
LIN {X 80.727,Y 56.242,Z 70.435,A 180.000,B 0.000,C 180.000} C_DIS
LIN {X 81.350,Y 56.242,Z 70.622,A 180.000,B 0.000,C 180.000} C_DIS
LIN {X 81.970,Y 56.242,Z 70.843,A 180.000,B 0.000,C 180.000} C_DIS
LIN {X 82.588,Y 56.242,Z 71.101,A 180.000,B 0.000,C 180.000} C_DIS
LIN {X 83.236,Y 56.242,Z 71.411,A 180.000,B 0.000,C 180.000} C_DIS
LIN {X 83.891,Y 56.242,Z 71.760,A 180.000,B 0.000,C 180.000} C_DIS
LIN {X 84.558,Y 56.242,Z 72.157,A 180.000,B 0.000,C 180.000} C_DIS
LIN {X 85.244,Y 56.242,Z 72.607,A 180.000,B 0.000,C 180.000} C_DIS
LIN {X 86.001,Y 56.242,Z 73.150,A 180.000,B 0.000,C 180.000} C_DIS
LIN {X 86.729,Y 56.242,Z 73.716,A 180.000,B 0.000,C 180.000} C_DIS
LIN {X 87.499,Y 56.242,Z 74.361,A 180.000,B 0.000,C 180.000} C_DIS
LIN {X 92.774,Y 56.242,Z 74.364,A 180.000,B 0.000,C 180.000} C_DIS
LIN {X 98.085,Y 56.242,Z 72.156,A 180.000,B 0.000,C 180.000} C_DIS
LIN {X 98.087,Y 56.242,Z 68.263,A 180.000,B 0.000,C 180.000} C_DIS
LIN {X 98.108,Y 56.242,Z 68.252,A 180.000,B 0.000,C 180.000} C_DIS
LIN {X 98.517,Y 56.242,Z 68.023,A 180.000,B 0.000,C 180.000} C_DIS
LIN {X 98.764,Y 56.242,Z 67.861,A 180.000,B 0.000,C 180.000} C_DIS
LIN {X 99.108,Y 56.242,Z 67.626,A 180.000,B 0.000,C 180.000} C_DIS
LIN {X 99.607,Y 56.242,Z 67.208,A 180.000,B 0.000,C 180.000} C_DIS
LIN {X 99.705,Y 56.242,Z 67.115,A 180.000,B 0.000,C 180.000} C_DIS
LIN {X 100.050,Y 56.242,Z 66.761,A 180.000,B 0.000,C 180.000} C_DIS
LIN {X 100.417,Y 56.242,Z 66.298,A 180.000,B 0.000,C 180.000} C_DIS
LIN {X 100.737,Y 56.242,Z 65.810,A 180.000,B 0.000,C 180.000} C_DIS
LIN {X 100.983,Y 56.242,Z 65.329,A 180.000,B 0.000,C 180.000} C_DIS
LIN {X 101.174,Y 56.242,Z 64.827,A 180.000,B 0.000,C 180.000} C_DIS
LIN {X 101.310,Y 56.242,Z 64.321,A 180.000,B 0.000,C 180.000} C_DIS
LIN {X 101.396,Y 56.242,Z 63.796,A 180.000,B 0.000,C 180.000} C_DIS
LIN {X 101.425,Y 56.242,Z 63.292,A 180.000,B 0.000,C 180.000} C_DIS
LIN {X 101.428,Y 56.242,Z 62.000,A 180.000,B 0.000,C 180.000} C_DIS
LIN {X 124.778,Y 56.242,Z 62.000,A 180.000,B 0.000,C 180.000} C_DIS
LIN {X 124.778,Y 56.242,Z 57.000,A 180.000,B 0.000,C 180.000} C_DIS
LIN {X 149.420,Y 56.242,Z 57.000,A 180.000,B 0.000,C 180.000} C_DIS
LIN {X 149.420,Y 56.242,Z 52.000,A 180.000,B 0.000,C 180.000} C_DIS
LIN {X 152.500,Y 56.242,Z 52.000,A 180.000,B 0.000,C 180.000} C_DIS
LIN {X 152.500,Y 56.242,Z 45.000,A 180.000,B 0.000,C 180.000} C_DIS
LIN {X 155.010,Y 56.242,Z 45.000,A 180.000,B 0.000,C 180.000} C_DIS
; Link Move Starts
LIN {X 155.120,Y 56.242,Z 45.026,A 180.000,B 0.000,C 180.000} C_DIS
LIN {X 155.230,Y 56.242,Z 45.051,A 180.000,B 0.000,C 180.000} C_DIS
LIN {X 155.771,Y 56.555,Z 45.051,A 180.000,B 0.000,C 180.000} C_DIS
LIN {X 155.771,Y 57.180,Z 45.051,A 180.000,B 0.000,C 180.000} C_DIS
LIN {X 155.230,Y 57.492,Z 45.051,A 180.000,B 0.000,C 180.000} C_DIS
LIN {X 155.120,Y 57.492,Z 45.026,A 180.000,B 0.000,C 180.000} C_DIS
LIN {X 155.010,Y 57.492,Z 45.000,A 180.000,B 0.000,C 180.000} C_DIS
; Cutting Move Starts
LIN {X 152.500,Y 57.492,Z 45.000,A 180.000,B 0.000,C 180.000} C_DIS
LIN {X 152.500,Y 57.492,Z 52.000,A 180.000,B 0.000,C 180.000} C_DIS
LIN {X 149.777,Y 57.492,Z 52.000,A 180.000,B 0.000,C 180.000} C_DIS
LIN {X 149.776,Y 57.492,Z 57.000,A 180.000,B 0.000,C 180.000} C_DIS
LIN {X 126.028,Y 57.492,Z 57.000,A 180.000,B 0.000,C 180.000} C_DIS
LIN {X 126.024,Y 57.492,Z 62.000,A 180.000,B 0.000,C 180.000} C_DIS
LIN {X 100.010,Y 57.492,Z 62.000,A 180.000,B 0.000,C 180.000} C_DIS
LIN {X 100.006,Y 57.492,Z 63.309,A 180.000,B 0.000,C 180.000} C_DIS
LIN {X 99.971,Y 57.492,Z 63.803,A 180.000,B 0.000,C 180.000} C_DIS
LIN {X 99.869,Y 57.492,Z 64.321,A 180.000,B 0.000,C 180.000} C_DIS
LIN {X 99.702,Y 57.492,Z 64.819,A 180.000,B 0.000,C 180.000} C_DIS
LIN {X 99.465,Y 57.492,Z 65.322,A 180.000,B 0.000,C 180.000} C_DIS
LIN {X 99.158,Y 57.492,Z 65.820,A 180.000,B 0.000,C 180.000} C_DIS
LIN {X 98.880,Y 57.492,Z 66.170,A 180.000,B 0.000,C 180.000} C_DIS
LIN {X 98.767,Y 57.492,Z 66.300,A 180.000,B 0.000,C 180.000} C_DIS
LIN {X 98.296,Y 57.492,Z 66.760,A 180.000,B 0.000,C 180.000} C_DIS
LIN {X 98.143,Y 57.492,Z 66.885,A 180.000,B 0.000,C 180.000} C_DIS
LIN {X 98.140,Y 57.492,Z 72.156,A 180.000,B 0.000,C 180.000} C_DIS
LIN {X 97.014,Y 57.492,Z 72.702,A 180.000,B 0.000,C 180.000} C_DIS
LIN {X 95.782,Y 57.492,Z 73.266,A 180.000,B 0.000,C 180.000} C_DIS
LIN {X 94.490,Y 57.492,Z 73.827,A 180.000,B 0.000,C 180.000} C_DIS
LIN {X 93.199,Y 57.492,Z 74.364,A 180.000,B 0.000,C 180.000} C_DIS
LIN {X 87.924,Y 57.492,Z 74.364,A 180.000,B 0.000,C 180.000} C_DIS
LIN {X 87.151,Y 57.492,Z 73.716,A 180.000,B 0.000,C 180.000} C_DIS
LIN {X 86.424,Y 57.492,Z 73.150,A 180.000,B 0.000,C 180.000} C_DIS
LIN {X 85.666,Y 57.492,Z 72.608,A 180.000,B 0.000,C 180.000} C_DIS
LIN {X 84.980,Y 57.492,Z 72.158,A 180.000,B 0.000,C 180.000} C_DIS
LIN {X 84.313,Y 57.492,Z 71.761,A 180.000,B 0.000,C 180.000} C_DIS
LIN {X 83.659,Y 57.492,Z 71.411,A 180.000,B 0.000,C 180.000} C_DIS
LIN {X 83.010,Y 57.492,Z 71.102,A 180.000,B 0.000,C 180.000} C_DIS
LIN {X 82.393,Y 57.492,Z 70.844,A 180.000,B 0.000,C 180.000} C_DIS
LIN {X 81.773,Y 57.492,Z 70.622,A 180.000,B 0.000,C 180.000} C_DIS
LIN {X 81.150,Y 57.492,Z 70.435,A 180.000,B 0.000,C 180.000} C_DIS
LIN {X 81.068,Y 57.492,Z 70.415,A 180.000,B 0.000,C 180.000} C_DIS
LIN {X 80.646,Y 57.492,Z 70.531,A 180.000,B 0.000,C 180.000} C_DIS
LIN {X 80.023,Y 57.492,Z 70.735,A 180.000,B 0.000,C 180.000} C_DIS
LIN {X 79.394,Y 57.492,Z 70.978,A 180.000,B 0.000,C 180.000} C_DIS
LIN {X 78.762,Y 57.492,Z 71.257,A 180.000,B 0.000,C 180.000} C_DIS
LIN {X 78.140,Y 57.492,Z 71.566,A 180.000,B 0.000,C 180.000} C_DIS
LIN {X 77.515,Y 57.492,Z 71.907,A 180.000,B 0.000,C 180.000} C_DIS
LIN {X 76.887,Y 57.492,Z 72.279,A 180.000,B 0.000,C 180.000} C_DIS
LIN {X 76.248,Y 57.492,Z 72.687,A 180.000,B 0.000,C 180.000} C_DIS
LIN {X 75.568,Y 57.492,Z 73.149,A 180.000,B 0.000,C 180.000} C_DIS
LIN {X 74.670,Y 57.492,Z 73.798,A 180.000,B 0.000,C 180.000} C_DIS
LIN {X 73.841,Y 57.492,Z 74.436,A 180.000,B 0.000,C 180.000} C_DIS
LIN {X 72.699,Y 57.492,Z 75.345,A 180.000,B 0.000,C 180.000} C_DIS
LIN {X 69.481,Y 57.492,Z 77.983,A 180.000,B 0.000,C 180.000} C_DIS
LIN {X 68.322,Y 57.492,Z 78.895,A 180.000,B 0.000,C 180.000} C_DIS
LIN {X 67.707,Y 57.492,Z 79.359,A 180.000,B 0.000,C 180.000} C_DIS
LIN {X 67.142,Y 57.492,Z 79.770,A 180.000,B 0.000,C 180.000} C_DIS
LIN {X 66.566,Y 57.492,Z 80.171,A 180.000,B 0.000,C 180.000} C_DIS
LIN {X 65.980,Y 57.492,Z 80.559,A 180.000,B 0.000,C 180.000} C_DIS
LIN {X 65.387,Y 57.492,Z 80.929,A 180.000,B 0.000,C 180.000} C_DIS
LIN {X 64.786,Y 57.492,Z 81.279,A 180.000,B 0.000,C 180.000} C_DIS
LIN {X 64.172,Y 57.492,Z 81.610,A 180.000,B 0.000,C 180.000} C_DIS
LIN {X 63.558,Y 57.492,Z 81.911,A 180.000,B 0.000,C 180.000} C_DIS
LIN {X 62.930,Y 57.492,Z 82.187,A 180.000,B 0.000,C 180.000} C_DIS
LIN {X 62.295,Y 57.492,Z 82.432,A 180.000,B 0.000,C 180.000} C_DIS
LIN {X 61.650,Y 57.492,Z 82.646,A 180.000,B 0.000,C 180.000} C_DIS
LIN {X 60.994,Y 57.492,Z 82.825,A 180.000,B 0.000,C 180.000} C_DIS
LIN {X 60.321,Y 57.492,Z 82.968,A 180.000,B 0.000,C 180.000} C_DIS
LIN {X 59.942,Y 57.492,Z 83.031,A 180.000,B 0.000,C 180.000} C_DIS
LIN {X 59.606,Y 57.492,Z 83.075,A 180.000,B 0.000,C 180.000} C_DIS
LIN {X 59.257,Y 57.492,Z 83.110,A 180.000,B 0.000,C 180.000} C_DIS
LIN {X 58.928,Y 57.492,Z 83.133,A 180.000,B 0.000,C 180.000} C_DIS
LIN {X 58.601,Y 57.492,Z 83.146,A 180.000,B 0.000,C 180.000} C_DIS
LIN {X 57.812,Y 57.492,Z 83.150,A 180.000,B 0.000,C 180.000} C_DIS
LIN {X 52.915,Y 57.492,Z 83.148,A 180.000,B 0.000,C 180.000} C_DIS
LIN {X 52.540,Y 57.492,Z 83.136,A 180.000,B 0.000,C 180.000} C_DIS
LIN {X 52.227,Y 57.492,Z 83.117,A 180.000,B 0.000,C 180.000} C_DIS
LIN {X 51.897,Y 57.492,Z 83.087,A 180.000,B 0.000,C 180.000} C_DIS
LIN {X 51.515,Y 57.492,Z 83.039,A 180.000,B 0.000,C 180.000} C_DIS
LIN {X 51.141,Y 57.492,Z 82.980,A 180.000,B 0.000,C 180.000} C_DIS
LIN {X 50.770,Y 57.492,Z 82.908,A 180.000,B 0.000,C 180.000} C_DIS
LIN {X 50.407,Y 57.492,Z 82.827,A 180.000,B 0.000,C 180.000} C_DIS
LIN {X 50.021,Y 57.492,Z 82.727,A 180.000,B 0.000,C 180.000} C_DIS
LIN {X 49.644,Y 57.492,Z 82.617,A 180.000,B 0.000,C 180.000} C_DIS
LIN {X 49.256,Y 57.492,Z 82.491,A 180.000,B 0.000,C 180.000} C_DIS
LIN {X 48.874,Y 57.492,Z 82.354,A 180.000,B 0.000,C 180.000} C_DIS
LIN {X 48.481,Y 57.492,Z 82.199,A 180.000,B 0.000,C 180.000} C_DIS
LIN {X 48.083,Y 57.492,Z 82.030,A 180.000,B 0.000,C 180.000} C_DIS
LIN {X 47.676,Y 57.492,Z 81.843,A 180.000,B 0.000,C 180.000} C_DIS
LIN {X 47.271,Y 57.492,Z 81.643,A 180.000,B 0.000,C 180.000} C_DIS
LIN {X 46.862,Y 57.492,Z 81.427,A 180.000,B 0.000,C 180.000} C_DIS
LIN {X 46.448,Y 57.492,Z 81.195,A 180.000,B 0.000,C 180.000} C_DIS
LIN {X 46.034,Y 57.492,Z 80.949,A 180.000,B 0.000,C 180.000} C_DIS
LIN {X 45.614,Y 57.492,Z 80.686,A 180.000,B 0.000,C 180.000} C_DIS
LIN {X 45.277,Y 57.492,Z 80.467,A 180.000,B 0.000,C 180.000} C_DIS
LIN {X 45.276,Y 57.492,Z 62.000,A 180.000,B 0.000,C 180.000} C_DIS
LIN {X 28.972,Y 57.492,Z 62.000,A 180.000,B 0.000,C 180.000} C_DIS
LIN {X 28.972,Y 57.492,Z 57.000,A 180.000,B 0.000,C 180.000} C_DIS
LIN {X 5.223,Y 57.492,Z 57.000,A 180.000,B 0.000,C 180.000} C_DIS
LIN {X 5.219,Y 57.492,Z 52.000,A 180.000,B 0.000,C 180.000} C_DIS
LIN {X 2.500,Y 57.492,Z 52.000,A 180.000,B 0.000,C 180.000} C_DIS
LIN {X 2.499,Y 57.492,Z 45.000,A 180.000,B 0.000,C 180.000} C_DIS
LIN {X -0.010,Y 57.492,Z 45.000,A 180.000,B 0.000,C 180.000} C_DIS
; Link Move Starts
LIN {X -0.120,Y 57.492,Z 45.026,A 180.000,B 0.000,C 180.000} C_DIS
LIN {X -0.230,Y 57.492,Z 45.051,A 180.000,B 0.000,C 180.000} C_DIS
LIN {X -0.771,Y 57.805,Z 45.051,A 180.000,B 0.000,C 180.000} C_DIS
LIN {X -0.771,Y 58.430,Z 45.051,A 180.000,B 0.000,C 180.000} C_DIS
LIN {X -0.230,Y 58.742,Z 45.051,A 180.000,B 0.000,C 180.000} C_DIS
LIN {X -0.120,Y 58.742,Z 45.026,A 180.000,B 0.000,C 180.000} C_DIS
LIN {X -0.010,Y 58.742,Z 45.000,A 180.000,B 0.000,C 180.000} C_DIS
; Cutting Move Starts
LIN {X 2.500,Y 58.742,Z 45.000,A 180.000,B 0.000,C 180.000} C_DIS
LIN {X 2.500,Y 58.742,Z 52.000,A 180.000,B 0.000,C 180.000} C_DIS
LIN {X 4.887,Y 58.742,Z 52.000,A 180.000,B 0.000,C 180.000} C_DIS
LIN {X 4.887,Y 58.742,Z 57.000,A 180.000,B 0.000,C 180.000} C_DIS
LIN {X 27.722,Y 58.742,Z 57.000,A 180.000,B 0.000,C 180.000} C_DIS
LIN {X 27.723,Y 58.742,Z 62.000,A 180.000,B 0.000,C 180.000} C_DIS
LIN {X 45.699,Y 58.742,Z 62.000,A 180.000,B 0.000,C 180.000} C_DIS
LIN {X 45.699,Y 58.742,Z 80.467,A 180.000,B 0.000,C 180.000} C_DIS
LIN {X 46.031,Y 58.742,Z 80.683,A 180.000,B 0.000,C 180.000} C_DIS
LIN {X 46.456,Y 58.742,Z 80.950,A 180.000,B 0.000,C 180.000} C_DIS
LIN {X 46.871,Y 58.742,Z 81.196,A 180.000,B 0.000,C 180.000} C_DIS
LIN {X 47.284,Y 58.742,Z 81.428,A 180.000,B 0.000,C 180.000} C_DIS
LIN {X 47.693,Y 58.742,Z 81.643,A 180.000,B 0.000,C 180.000} C_DIS
LIN {X 48.098,Y 58.742,Z 81.843,A 180.000,B 0.000,C 180.000} C_DIS
LIN {X 48.505,Y 58.742,Z 82.030,A 180.000,B 0.000,C 180.000} C_DIS
LIN {X 48.902,Y 58.742,Z 82.199,A 180.000,B 0.000,C 180.000} C_DIS
LIN {X 49.296,Y 58.742,Z 82.354,A 180.000,B 0.000,C 180.000} C_DIS
LIN {X 49.677,Y 58.742,Z 82.491,A 180.000,B 0.000,C 180.000} C_DIS
LIN {X 50.066,Y 58.742,Z 82.617,A 180.000,B 0.000,C 180.000} C_DIS
LIN {X 50.443,Y 58.742,Z 82.727,A 180.000,B 0.000,C 180.000} C_DIS
LIN {X 50.829,Y 58.742,Z 82.827,A 180.000,B 0.000,C 180.000} C_DIS
LIN {X 51.191,Y 58.742,Z 82.908,A 180.000,B 0.000,C 180.000} C_DIS
LIN {X 51.562,Y 58.742,Z 82.980,A 180.000,B 0.000,C 180.000} C_DIS
LIN {X 51.936,Y 58.742,Z 83.039,A 180.000,B 0.000,C 180.000} C_DIS
LIN {X 52.318,Y 58.742,Z 83.087,A 180.000,B 0.000,C 180.000} C_DIS
LIN {X 52.649,Y 58.742,Z 83.117,A 180.000,B 0.000,C 180.000} C_DIS
LIN {X 52.961,Y 58.742,Z 83.136,A 180.000,B 0.000,C 180.000} C_DIS
LIN {X 53.336,Y 58.742,Z 83.148,A 180.000,B 0.000,C 180.000} C_DIS
LIN {X 58.234,Y 58.742,Z 83.150,A 180.000,B 0.000,C 180.000} C_DIS
LIN {X 59.022,Y 58.742,Z 83.146,A 180.000,B 0.000,C 180.000} C_DIS
LIN {X 59.349,Y 58.742,Z 83.133,A 180.000,B 0.000,C 180.000} C_DIS
LIN {X 59.679,Y 58.742,Z 83.110,A 180.000,B 0.000,C 180.000} C_DIS
LIN {X 60.027,Y 58.742,Z 83.075,A 180.000,B 0.000,C 180.000} C_DIS
LIN {X 60.363,Y 58.742,Z 83.031,A 180.000,B 0.000,C 180.000} C_DIS
LIN {X 60.743,Y 58.742,Z 82.968,A 180.000,B 0.000,C 180.000} C_DIS
LIN {X 61.416,Y 58.742,Z 82.825,A 180.000,B 0.000,C 180.000} C_DIS
LIN {X 62.071,Y 58.742,Z 82.646,A 180.000,B 0.000,C 180.000} C_DIS
LIN {X 62.717,Y 58.742,Z 82.432,A 180.000,B 0.000,C 180.000} C_DIS
LIN {X 63.352,Y 58.742,Z 82.187,A 180.000,B 0.000,C 180.000} C_DIS
LIN {X 63.980,Y 58.742,Z 81.911,A 180.000,B 0.000,C 180.000} C_DIS
LIN {X 64.593,Y 58.742,Z 81.610,A 180.000,B 0.000,C 180.000} C_DIS
LIN {X 65.207,Y 58.742,Z 81.279,A 180.000,B 0.000,C 180.000} C_DIS
LIN {X 65.808,Y 58.742,Z 80.929,A 180.000,B 0.000,C 180.000} C_DIS
LIN {X 66.402,Y 58.742,Z 80.559,A 180.000,B 0.000,C 180.000} C_DIS
LIN {X 66.987,Y 58.742,Z 80.171,A 180.000,B 0.000,C 180.000} C_DIS
LIN {X 67.563,Y 58.742,Z 79.770,A 180.000,B 0.000,C 180.000} C_DIS
LIN {X 68.128,Y 58.742,Z 79.359,A 180.000,B 0.000,C 180.000} C_DIS
LIN {X 68.744,Y 58.742,Z 78.896,A 180.000,B 0.000,C 180.000} C_DIS
LIN {X 69.903,Y 58.742,Z 77.983,A 180.000,B 0.000,C 180.000} C_DIS
LIN {X 73.121,Y 58.742,Z 75.345,A 180.000,B 0.000,C 180.000} C_DIS
LIN {X 74.263,Y 58.742,Z 74.436,A 180.000,B 0.000,C 180.000} C_DIS
LIN {X 75.092,Y 58.742,Z 73.798,A 180.000,B 0.000,C 180.000} C_DIS
LIN {X 75.990,Y 58.742,Z 73.149,A 180.000,B 0.000,C 180.000} C_DIS
LIN {X 76.669,Y 58.742,Z 72.687,A 180.000,B 0.000,C 180.000} C_DIS
LIN {X 77.308,Y 58.742,Z 72.279,A 180.000,B 0.000,C 180.000} C_DIS
LIN {X 77.936,Y 58.742,Z 71.907,A 180.000,B 0.000,C 180.000} C_DIS
LIN {X 78.561,Y 58.742,Z 71.566,A 180.000,B 0.000,C 180.000} C_DIS
LIN {X 79.183,Y 58.742,Z 71.257,A 180.000,B 0.000,C 180.000} C_DIS
LIN {X 79.816,Y 58.742,Z 70.978,A 180.000,B 0.000,C 180.000} C_DIS
LIN {X 80.444,Y 58.742,Z 70.735,A 180.000,B 0.000,C 180.000} C_DIS
LIN {X 81.067,Y 58.742,Z 70.531,A 180.000,B 0.000,C 180.000} C_DIS
LIN {X 81.488,Y 58.742,Z 70.415,A 180.000,B 0.000,C 180.000} C_DIS
LIN {X 81.594,Y 58.742,Z 70.441,A 180.000,B 0.000,C 180.000} C_DIS
LIN {X 82.202,Y 58.742,Z 70.625,A 180.000,B 0.000,C 180.000} C_DIS
LIN {X 82.813,Y 58.742,Z 70.843,A 180.000,B 0.000,C 180.000} C_DIS
LIN {X 83.431,Y 58.742,Z 71.101,A 180.000,B 0.000,C 180.000} C_DIS
LIN {X 84.079,Y 58.742,Z 71.411,A 180.000,B 0.000,C 180.000} C_DIS
LIN {X 84.734,Y 58.742,Z 71.760,A 180.000,B 0.000,C 180.000} C_DIS
LIN {X 85.401,Y 58.742,Z 72.157,A 180.000,B 0.000,C 180.000} C_DIS
LIN {X 86.087,Y 58.742,Z 72.607,A 180.000,B 0.000,C 180.000} C_DIS
LIN {X 86.844,Y 58.742,Z 73.150,A 180.000,B 0.000,C 180.000} C_DIS
LIN {X 87.572,Y 58.742,Z 73.715,A 180.000,B 0.000,C 180.000} C_DIS
LIN {X 88.346,Y 58.742,Z 74.364,A 180.000,B 0.000,C 180.000} C_DIS
LIN {X 93.421,Y 58.742,Z 74.364,A 180.000,B 0.000,C 180.000} C_DIS
LIN {X 93.465,Y 58.742,Z 74.345,A 180.000,B 0.000,C 180.000} C_DIS
LIN {X 94.574,Y 58.742,Z 73.804,A 180.000,B 0.000,C 180.000} C_DIS
LIN {X 95.538,Y 58.742,Z 73.304,A 180.000,B 0.000,C 180.000} C_DIS
LIN {X 96.341,Y 58.742,Z 72.858,A 180.000,B 0.000,C 180.000} C_DIS
LIN {X 96.981,Y 58.742,Z 72.474,A 180.000,B 0.000,C 180.000} C_DIS
LIN {X 97.464,Y 58.742,Z 72.156,A 180.000,B 0.000,C 180.000} C_DIS
LIN {X 97.465,Y 58.742,Z 64.916,A 180.000,B 0.000,C 180.000} C_DIS
LIN {X 97.534,Y 58.742,Z 64.812,A 180.000,B 0.000,C 180.000} C_DIS
LIN {X 97.774,Y 58.742,Z 64.297,A 180.000,B 0.000,C 180.000} C_DIS
LIN {X 97.915,Y 58.742,Z 63.790,A 180.000,B 0.000,C 180.000} C_DIS
LIN {X 97.962,Y 58.742,Z 63.281,A 180.000,B 0.000,C 180.000} C_DIS
LIN {X 97.965,Y 58.742,Z 62.000,A 180.000,B 0.000,C 180.000} C_DIS
LIN {X 127.277,Y 58.742,Z 62.000,A 180.000,B 0.000,C 180.000} C_DIS
LIN {X 127.278,Y 58.742,Z 57.000,A 180.000,B 0.000,C 180.000} C_DIS
LIN {X 150.112,Y 58.742,Z 57.000,A 180.000,B 0.000,C 180.000} C_DIS
LIN {X 150.113,Y 58.742,Z 52.000,A 180.000,B 0.000,C 180.000} C_DIS
LIN {X 152.500,Y 58.742,Z 52.000,A 180.000,B 0.000,C 180.000} C_DIS
LIN {X 152.500,Y 58.742,Z 45.000,A 180.000,B 0.000,C 180.000} C_DIS
LIN {X 155.010,Y 58.742,Z 45.000,A 180.000,B 0.000,C 180.000} C_DIS
; Link Move Starts
LIN {X 155.120,Y 58.742,Z 45.026,A 180.000,B 0.000,C 180.000} C_DIS
LIN {X 155.230,Y 58.742,Z 45.051,A 180.000,B 0.000,C 180.000} C_DIS
LIN {X 155.771,Y 59.054,Z 45.051,A 180.000,B 0.000,C 180.000} C_DIS
LIN {X 155.771,Y 59.679,Z 45.051,A 180.000,B 0.000,C 180.000} C_DIS
LIN {X 155.230,Y 59.992,Z 45.051,A 180.000,B 0.000,C 180.000} C_DIS
LIN {X 155.120,Y 59.992,Z 45.026,A 180.000,B 0.000,C 180.000} C_DIS
LIN {X 155.010,Y 59.992,Z 45.000,A 180.000,B 0.000,C 180.000} C_DIS
; Cutting Move Starts
LIN {X 152.500,Y 59.992,Z 45.000,A 180.000,B 0.000,C 180.000} C_DIS
LIN {X 152.500,Y 59.992,Z 52.000,A 180.000,B 0.000,C 180.000} C_DIS
LIN {X 150.427,Y 59.992,Z 52.000,A 180.000,B 0.000,C 180.000} C_DIS
LIN {X 150.427,Y 59.992,Z 57.000,A 180.000,B 0.000,C 180.000} C_DIS
LIN {X 128.527,Y 59.992,Z 57.000,A 180.000,B 0.000,C 180.000} C_DIS
LIN {X 128.526,Y 59.992,Z 62.000,A 180.000,B 0.000,C 180.000} C_DIS
LIN {X 94.576,Y 59.992,Z 62.000,A 180.000,B 0.000,C 180.000} C_DIS
LIN {X 94.572,Y 59.992,Z 73.081,A 180.000,B 0.000,C 180.000} C_DIS
LIN {X 94.537,Y 59.992,Z 73.171,A 180.000,B 0.000,C 180.000} C_DIS
LIN {X 94.443,Y 59.992,Z 73.302,A 180.000,B 0.000,C 180.000} C_DIS
LIN {X 94.263,Y 59.992,Z 73.482,A 180.000,B 0.000,C 180.000} C_DIS
LIN {X 93.988,Y 59.992,Z 73.707,A 180.000,B 0.000,C 180.000} C_DIS
LIN {X 93.592,Y 59.992,Z 73.987,A 180.000,B 0.000,C 180.000} C_DIS
LIN {X 93.052,Y 59.992,Z 74.330,A 180.000,B 0.000,C 180.000} C_DIS
LIN {X 92.992,Y 59.992,Z 74.364,A 180.000,B 0.000,C 180.000} C_DIS
LIN {X 88.861,Y 59.992,Z 74.361,A 180.000,B 0.000,C 180.000} C_DIS
LIN {X 87.833,Y 59.992,Z 73.567,A 180.000,B 0.000,C 180.000} C_DIS
LIN {X 87.030,Y 59.992,Z 72.974,A 180.000,B 0.000,C 180.000} C_DIS
LIN {X 86.273,Y 59.992,Z 72.447,A 180.000,B 0.000,C 180.000} C_DIS
LIN {X 85.585,Y 59.992,Z 72.012,A 180.000,B 0.000,C 180.000} C_DIS
LIN {X 84.905,Y 59.992,Z 71.622,A 180.000,B 0.000,C 180.000} C_DIS
LIN {X 84.256,Y 59.992,Z 71.289,A 180.000,B 0.000,C 180.000} C_DIS
LIN {X 83.631,Y 59.992,Z 71.005,A 180.000,B 0.000,C 180.000} C_DIS
LIN {X 82.998,Y 59.992,Z 70.755,A 180.000,B 0.000,C 180.000} C_DIS
LIN {X 82.383,Y 59.992,Z 70.547,A 180.000,B 0.000,C 180.000} C_DIS
LIN {X 81.913,Y 59.992,Z 70.414,A 180.000,B 0.000,C 180.000} C_DIS
LIN {X 81.489,Y 59.992,Z 70.531,A 180.000,B 0.000,C 180.000} C_DIS
LIN {X 80.866,Y 59.992,Z 70.735,A 180.000,B 0.000,C 180.000} C_DIS
LIN {X 80.237,Y 59.992,Z 70.978,A 180.000,B 0.000,C 180.000} C_DIS
LIN {X 79.605,Y 59.992,Z 71.257,A 180.000,B 0.000,C 180.000} C_DIS
LIN {X 78.983,Y 59.992,Z 71.566,A 180.000,B 0.000,C 180.000} C_DIS
LIN {X 78.358,Y 59.992,Z 71.907,A 180.000,B 0.000,C 180.000} C_DIS
LIN {X 77.730,Y 59.992,Z 72.279,A 180.000,B 0.000,C 180.000} C_DIS
LIN {X 77.091,Y 59.992,Z 72.687,A 180.000,B 0.000,C 180.000} C_DIS
LIN {X 76.411,Y 59.992,Z 73.149,A 180.000,B 0.000,C 180.000} C_DIS
LIN {X 75.514,Y 59.992,Z 73.798,A 180.000,B 0.000,C 180.000} C_DIS
LIN {X 74.684,Y 59.992,Z 74.436,A 180.000,B 0.000,C 180.000} C_DIS
LIN {X 73.543,Y 59.992,Z 75.345,A 180.000,B 0.000,C 180.000} C_DIS
LIN {X 70.325,Y 59.992,Z 77.983,A 180.000,B 0.000,C 180.000} C_DIS
LIN {X 69.166,Y 59.992,Z 78.895,A 180.000,B 0.000,C 180.000} C_DIS
LIN {X 68.550,Y 59.992,Z 79.359,A 180.000,B 0.000,C 180.000} C_DIS
LIN {X 67.985,Y 59.992,Z 79.770,A 180.000,B 0.000,C 180.000} C_DIS
LIN {X 67.409,Y 59.992,Z 80.171,A 180.000,B 0.000,C 180.000} C_DIS
LIN {X 66.824,Y 59.992,Z 80.559,A 180.000,B 0.000,C 180.000} C_DIS
LIN {X 66.230,Y 59.992,Z 80.929,A 180.000,B 0.000,C 180.000} C_DIS
LIN {X 65.629,Y 59.992,Z 81.279,A 180.000,B 0.000,C 180.000} C_DIS
LIN {X 65.015,Y 59.992,Z 81.610,A 180.000,B 0.000,C 180.000} C_DIS
LIN {X 64.402,Y 59.992,Z 81.911,A 180.000,B 0.000,C 180.000} C_DIS
LIN {X 63.773,Y 59.992,Z 82.187,A 180.000,B 0.000,C 180.000} C_DIS
LIN {X 63.138,Y 59.992,Z 82.432,A 180.000,B 0.000,C 180.000} C_DIS
LIN {X 62.493,Y 59.992,Z 82.646,A 180.000,B 0.000,C 180.000} C_DIS
LIN {X 61.838,Y 59.992,Z 82.825,A 180.000,B 0.000,C 180.000} C_DIS
LIN {X 61.164,Y 59.992,Z 82.968,A 180.000,B 0.000,C 180.000} C_DIS
LIN {X 60.785,Y 59.992,Z 83.031,A 180.000,B 0.000,C 180.000} C_DIS
LIN {X 60.449,Y 59.992,Z 83.075,A 180.000,B 0.000,C 180.000} C_DIS
LIN {X 60.100,Y 59.992,Z 83.110,A 180.000,B 0.000,C 180.000} C_DIS
LIN {X 59.771,Y 59.992,Z 83.133,A 180.000,B 0.000,C 180.000} C_DIS
LIN {X 59.444,Y 59.992,Z 83.146,A 180.000,B 0.000,C 180.000} C_DIS
LIN {X 58.655,Y 59.992,Z 83.150,A 180.000,B 0.000,C 180.000} C_DIS
LIN {X 53.758,Y 59.992,Z 83.148,A 180.000,B 0.000,C 180.000} C_DIS
LIN {X 53.383,Y 59.992,Z 83.136,A 180.000,B 0.000,C 180.000} C_DIS
LIN {X 53.071,Y 59.992,Z 83.117,A 180.000,B 0.000,C 180.000} C_DIS
LIN {X 52.740,Y 59.992,Z 83.087,A 180.000,B 0.000,C 180.000} C_DIS
LIN {X 52.358,Y 59.992,Z 83.039,A 180.000,B 0.000,C 180.000} C_DIS
LIN {X 51.984,Y 59.992,Z 82.980,A 180.000,B 0.000,C 180.000} C_DIS
LIN {X 51.613,Y 59.992,Z 82.908,A 180.000,B 0.000,C 180.000} C_DIS
LIN {X 51.251,Y 59.992,Z 82.827,A 180.000,B 0.000,C 180.000} C_DIS
LIN {X 50.865,Y 59.992,Z 82.727,A 180.000,B 0.000,C 180.000} C_DIS
LIN {X 50.488,Y 59.992,Z 82.617,A 180.000,B 0.000,C 180.000} C_DIS
LIN {X 50.099,Y 59.992,Z 82.491,A 180.000,B 0.000,C 180.000} C_DIS
LIN {X 49.718,Y 59.992,Z 82.354,A 180.000,B 0.000,C 180.000} C_DIS
LIN {X 49.324,Y 59.992,Z 82.199,A 180.000,B 0.000,C 180.000} C_DIS
LIN {X 48.927,Y 59.992,Z 82.030,A 180.000,B 0.000,C 180.000} C_DIS
LIN {X 48.520,Y 59.992,Z 81.843,A 180.000,B 0.000,C 180.000} C_DIS
LIN {X 48.115,Y 59.992,Z 81.643,A 180.000,B 0.000,C 180.000} C_DIS
LIN {X 47.706,Y 59.992,Z 81.427,A 180.000,B 0.000,C 180.000} C_DIS
LIN {X 47.292,Y 59.992,Z 81.195,A 180.000,B 0.000,C 180.000} C_DIS
LIN {X 46.877,Y 59.992,Z 80.950,A 180.000,B 0.000,C 180.000} C_DIS
LIN {X 46.457,Y 59.992,Z 80.686,A 180.000,B 0.000,C 180.000} C_DIS
LIN {X 46.121,Y 59.992,Z 80.467,A 180.000,B 0.000,C 180.000} C_DIS
LIN {X 46.121,Y 59.992,Z 62.000,A 180.000,B 0.000,C 180.000} C_DIS
LIN {X 26.473,Y 59.992,Z 62.000,A 180.000,B 0.000,C 180.000} C_DIS
LIN {X 26.473,Y 59.992,Z 57.000,A 180.000,B 0.000,C 180.000} C_DIS
LIN {X 4.573,Y 59.992,Z 57.000,A 180.000,B 0.000,C 180.000} C_DIS
LIN {X 4.573,Y 59.992,Z 52.000,A 180.000,B 0.000,C 180.000} C_DIS
LIN {X 2.500,Y 59.992,Z 52.000,A 180.000,B 0.000,C 180.000} C_DIS
LIN {X 2.500,Y 59.992,Z 45.000,A 180.000,B 0.000,C 180.000} C_DIS
LIN {X -0.010,Y 59.992,Z 45.000,A 180.000,B 0.000,C 180.000} C_DIS
; Link Move Starts
LIN {X -0.120,Y 59.992,Z 45.026,A 180.000,B 0.000,C 180.000} C_DIS
LIN {X -0.230,Y 59.992,Z 45.051,A 180.000,B 0.000,C 180.000} C_DIS
LIN {X -0.771,Y 60.304,Z 45.051,A 180.000,B 0.000,C 180.000} C_DIS
LIN {X -0.771,Y 60.929,Z 45.051,A 180.000,B 0.000,C 180.000} C_DIS
LIN {X -0.230,Y 61.242,Z 45.051,A 180.000,B 0.000,C 180.000} C_DIS
LIN {X -0.120,Y 61.242,Z 45.026,A 180.000,B 0.000,C 180.000} C_DIS
LIN {X -0.010,Y 61.242,Z 45.000,A 180.000,B 0.000,C 180.000} C_DIS
; Cutting Move Starts
LIN {X 2.500,Y 61.242,Z 45.000,A 180.000,B 0.000,C 180.000} C_DIS
LIN {X 2.500,Y 61.242,Z 52.000,A 180.000,B 0.000,C 180.000} C_DIS
LIN {X 4.288,Y 61.242,Z 52.000,A 180.000,B 0.000,C 180.000} C_DIS
LIN {X 4.288,Y 61.242,Z 57.000,A 180.000,B 0.000,C 180.000} C_DIS
LIN {X 25.223,Y 61.242,Z 57.000,A 180.000,B 0.000,C 180.000} C_DIS
LIN {X 25.223,Y 61.242,Z 62.000,A 180.000,B 0.000,C 180.000} C_DIS
LIN {X 46.541,Y 61.242,Z 62.000,A 180.000,B 0.000,C 180.000} C_DIS
LIN {X 46.542,Y 61.242,Z 80.467,A 180.000,B 0.000,C 180.000} C_DIS
LIN {X 46.874,Y 61.242,Z 80.683,A 180.000,B 0.000,C 180.000} C_DIS
LIN {X 47.299,Y 61.242,Z 80.950,A 180.000,B 0.000,C 180.000} C_DIS
LIN {X 47.714,Y 61.242,Z 81.196,A 180.000,B 0.000,C 180.000} C_DIS
LIN {X 48.128,Y 61.242,Z 81.428,A 180.000,B 0.000,C 180.000} C_DIS
LIN {X 48.537,Y 61.242,Z 81.643,A 180.000,B 0.000,C 180.000} C_DIS
LIN {X 48.942,Y 61.242,Z 81.843,A 180.000,B 0.000,C 180.000} C_DIS
LIN {X 49.349,Y 61.242,Z 82.030,A 180.000,B 0.000,C 180.000} C_DIS
LIN {X 49.746,Y 61.242,Z 82.199,A 180.000,B 0.000,C 180.000} C_DIS
LIN {X 50.139,Y 61.242,Z 82.354,A 180.000,B 0.000,C 180.000} C_DIS
LIN {X 50.521,Y 61.242,Z 82.491,A 180.000,B 0.000,C 180.000} C_DIS
LIN {X 50.909,Y 61.242,Z 82.617,A 180.000,B 0.000,C 180.000} C_DIS
LIN {X 51.286,Y 61.242,Z 82.727,A 180.000,B 0.000,C 180.000} C_DIS
LIN {X 51.672,Y 61.242,Z 82.827,A 180.000,B 0.000,C 180.000} C_DIS
LIN {X 52.035,Y 61.242,Z 82.908,A 180.000,B 0.000,C 180.000} C_DIS
LIN {X 52.406,Y 61.242,Z 82.980,A 180.000,B 0.000,C 180.000} C_DIS
LIN {X 52.779,Y 61.242,Z 83.039,A 180.000,B 0.000,C 180.000} C_DIS
LIN {X 53.162,Y 61.242,Z 83.087,A 180.000,B 0.000,C 180.000} C_DIS
LIN {X 53.492,Y 61.242,Z 83.117,A 180.000,B 0.000,C 180.000} C_DIS
LIN {X 53.805,Y 61.242,Z 83.136,A 180.000,B 0.000,C 180.000} C_DIS
LIN {X 54.179,Y 61.242,Z 83.148,A 180.000,B 0.000,C 180.000} C_DIS
LIN {X 59.077,Y 61.242,Z 83.150,A 180.000,B 0.000,C 180.000} C_DIS
LIN {X 59.866,Y 61.242,Z 83.146,A 180.000,B 0.000,C 180.000} C_DIS
LIN {X 60.192,Y 61.242,Z 83.133,A 180.000,B 0.000,C 180.000} C_DIS
LIN {X 60.522,Y 61.242,Z 83.110,A 180.000,B 0.000,C 180.000} C_DIS
LIN {X 60.871,Y 61.242,Z 83.075,A 180.000,B 0.000,C 180.000} C_DIS
LIN {X 61.207,Y 61.242,Z 83.031,A 180.000,B 0.000,C 180.000} C_DIS
LIN {X 61.586,Y 61.242,Z 82.968,A 180.000,B 0.000,C 180.000} C_DIS
LIN {X 62.259,Y 61.242,Z 82.825,A 180.000,B 0.000,C 180.000} C_DIS
LIN {X 62.915,Y 61.242,Z 82.646,A 180.000,B 0.000,C 180.000} C_DIS
LIN {X 63.560,Y 61.242,Z 82.432,A 180.000,B 0.000,C 180.000} C_DIS
LIN {X 64.195,Y 61.242,Z 82.187,A 180.000,B 0.000,C 180.000} C_DIS
LIN {X 64.823,Y 61.242,Z 81.911,A 180.000,B 0.000,C 180.000} C_DIS
LIN {X 65.437,Y 61.242,Z 81.610,A 180.000,B 0.000,C 180.000} C_DIS
LIN {X 66.051,Y 61.242,Z 81.279,A 180.000,B 0.000,C 180.000} C_DIS
LIN {X 66.652,Y 61.242,Z 80.929,A 180.000,B 0.000,C 180.000} C_DIS
LIN {X 67.245,Y 61.242,Z 80.559,A 180.000,B 0.000,C 180.000} C_DIS
LIN {X 67.831,Y 61.242,Z 80.171,A 180.000,B 0.000,C 180.000} C_DIS
LIN {X 68.406,Y 61.242,Z 79.770,A 180.000,B 0.000,C 180.000} C_DIS
LIN {X 68.972,Y 61.242,Z 79.359,A 180.000,B 0.000,C 180.000} C_DIS
LIN {X 69.587,Y 61.242,Z 78.896,A 180.000,B 0.000,C 180.000} C_DIS
LIN {X 70.746,Y 61.242,Z 77.983,A 180.000,B 0.000,C 180.000} C_DIS
LIN {X 73.964,Y 61.242,Z 75.345,A 180.000,B 0.000,C 180.000} C_DIS
LIN {X 75.106,Y 61.242,Z 74.436,A 180.000,B 0.000,C 180.000} C_DIS
LIN {X 75.935,Y 61.242,Z 73.798,A 180.000,B 0.000,C 180.000} C_DIS
LIN {X 76.833,Y 61.242,Z 73.149,A 180.000,B 0.000,C 180.000} C_DIS
LIN {X 77.512,Y 61.242,Z 72.687,A 180.000,B 0.000,C 180.000} C_DIS
LIN {X 78.152,Y 61.242,Z 72.279,A 180.000,B 0.000,C 180.000} C_DIS
LIN {X 78.779,Y 61.242,Z 71.907,A 180.000,B 0.000,C 180.000} C_DIS
LIN {X 79.404,Y 61.242,Z 71.566,A 180.000,B 0.000,C 180.000} C_DIS
LIN {X 80.027,Y 61.242,Z 71.257,A 180.000,B 0.000,C 180.000} C_DIS
LIN {X 80.659,Y 61.242,Z 70.978,A 180.000,B 0.000,C 180.000} C_DIS
LIN {X 81.287,Y 61.242,Z 70.735,A 180.000,B 0.000,C 180.000} C_DIS
LIN {X 81.911,Y 61.242,Z 70.531,A 180.000,B 0.000,C 180.000} C_DIS
LIN {X 82.334,Y 61.242,Z 70.414,A 180.000,B 0.000,C 180.000} C_DIS
LIN {X 82.954,Y 61.242,Z 70.595,A 180.000,B 0.000,C 180.000} C_DIS
LIN {X 83.463,Y 61.242,Z 70.769,A 180.000,B 0.000,C 180.000} C_DIS
LIN {X 84.089,Y 61.242,Z 71.010,A 180.000,B 0.000,C 180.000} C_DIS
LIN {X 84.692,Y 61.242,Z 71.268,A 180.000,B 0.000,C 180.000} C_DIS
LIN {X 85.414,Y 61.242,Z 71.603,A 180.000,B 0.000,C 180.000} C_DIS
LIN {X 86.213,Y 61.242,Z 72.000,A 180.000,B 0.000,C 180.000} C_DIS
LIN {X 88.270,Y 61.242,Z 73.081,A 180.000,B 0.000,C 180.000} C_DIS
LIN {X 89.012,Y 61.242,Z 73.450,A 180.000,B 0.000,C 180.000} C_DIS
LIN {X 89.475,Y 61.242,Z 73.654,A 180.000,B 0.000,C 180.000} C_DIS
LIN {X 89.843,Y 61.242,Z 73.794,A 180.000,B 0.000,C 180.000} C_DIS
LIN {X 90.132,Y 61.242,Z 73.877,A 180.000,B 0.000,C 180.000} C_DIS
LIN {X 90.354,Y 61.242,Z 73.915,A 180.000,B 0.000,C 180.000} C_DIS
LIN {X 90.525,Y 61.242,Z 73.918,A 180.000,B 0.000,C 180.000} C_DIS
LIN {X 90.642,Y 61.242,Z 73.897,A 180.000,B 0.000,C 180.000} C_DIS
LIN {X 90.734,Y 61.242,Z 73.856,A 180.000,B 0.000,C 180.000} C_DIS
LIN {X 90.799,Y 61.242,Z 73.799,A 180.000,B 0.000,C 180.000} C_DIS
LIN {X 90.843,Y 61.242,Z 73.723,A 180.000,B 0.000,C 180.000} C_DIS
LIN {X 90.868,Y 61.242,Z 73.624,A 180.000,B 0.000,C 180.000} C_DIS
LIN {X 90.871,Y 61.242,Z 62.000,A 180.000,B 0.000,C 180.000} C_DIS
LIN {X 129.775,Y 61.242,Z 62.000,A 180.000,B 0.000,C 180.000} C_DIS
LIN {X 129.777,Y 61.242,Z 57.000,A 180.000,B 0.000,C 180.000} C_DIS
LIN {X 150.709,Y 61.242,Z 57.000,A 180.000,B 0.000,C 180.000} C_DIS
LIN {X 150.712,Y 61.242,Z 52.000,A 180.000,B 0.000,C 180.000} C_DIS
LIN {X 152.500,Y 61.242,Z 52.000,A 180.000,B 0.000,C 180.000} C_DIS
LIN {X 152.500,Y 61.242,Z 45.000,A 180.000,B 0.000,C 180.000} C_DIS
LIN {X 155.010,Y 61.242,Z 45.000,A 180.000,B 0.000,C 180.000} C_DIS
; Link Move Starts
LIN {X 155.120,Y 61.242,Z 45.026,A 180.000,B 0.000,C 180.000} C_DIS
LIN {X 155.230,Y 61.242,Z 45.051,A 180.000,B 0.000,C 180.000} C_DIS
LIN {X 155.771,Y 61.554,Z 45.051,A 180.000,B 0.000,C 180.000} C_DIS
LIN {X 155.771,Y 62.179,Z 45.051,A 180.000,B 0.000,C 180.000} C_DIS
LIN {X 155.230,Y 62.492,Z 45.051,A 180.000,B 0.000,C 180.000} C_DIS
LIN {X 155.120,Y 62.492,Z 45.026,A 180.000,B 0.000,C 180.000} C_DIS
LIN {X 155.010,Y 62.492,Z 45.000,A 180.000,B 0.000,C 180.000} C_DIS
; Cutting Move Starts
LIN {X 152.500,Y 62.492,Z 45.000,A 180.000,B 0.000,C 180.000} C_DIS
LIN {X 152.500,Y 62.492,Z 52.000,A 180.000,B 0.000,C 180.000} C_DIS
LIN {X 150.978,Y 62.492,Z 52.000,A 180.000,B 0.000,C 180.000} C_DIS
LIN {X 150.978,Y 62.492,Z 57.000,A 180.000,B 0.000,C 180.000} C_DIS
LIN {X 131.027,Y 62.492,Z 57.000,A 180.000,B 0.000,C 180.000} C_DIS
LIN {X 131.027,Y 62.492,Z 62.000,A 180.000,B 0.000,C 180.000} C_DIS
LIN {X 87.166,Y 62.492,Z 62.000,A 180.000,B 0.000,C 180.000} C_DIS
LIN {X 87.161,Y 62.492,Z 71.065,A 180.000,B 0.000,C 180.000} C_DIS
LIN {X 87.129,Y 62.492,Z 71.122,A 180.000,B 0.000,C 180.000} C_DIS
LIN {X 87.063,Y 62.492,Z 71.172,A 180.000,B 0.000,C 180.000} C_DIS
LIN {X 86.957,Y 62.492,Z 71.206,A 180.000,B 0.000,C 180.000} C_DIS
LIN {X 86.804,Y 62.492,Z 71.222,A 180.000,B 0.000,C 180.000} C_DIS
LIN {X 86.555,Y 62.492,Z 71.213,A 180.000,B 0.000,C 180.000} C_DIS
LIN {X 86.216,Y 62.492,Z 71.165,A 180.000,B 0.000,C 180.000} C_DIS
LIN {X 85.661,Y 62.492,Z 71.050,A 180.000,B 0.000,C 180.000} C_DIS
LIN {X 84.312,Y 62.492,Z 70.707,A 180.000,B 0.000,C 180.000} C_DIS
LIN {X 83.451,Y 62.492,Z 70.498,A 180.000,B 0.000,C 180.000} C_DIS
LIN {X 82.751,Y 62.492,Z 70.348,A 180.000,B 0.000,C 180.000} C_DIS
LIN {X 82.192,Y 62.492,Z 70.518,A 180.000,B 0.000,C 180.000} C_DIS
LIN {X 81.620,Y 62.492,Z 70.726,A 180.000,B 0.000,C 180.000} C_DIS
LIN {X 81.040,Y 62.492,Z 70.968,A 180.000,B 0.000,C 180.000} C_DIS
LIN {X 80.450,Y 62.492,Z 71.244,A 180.000,B 0.000,C 180.000} C_DIS
LIN {X 79.846,Y 62.492,Z 71.552,A 180.000,B 0.000,C 180.000} C_DIS
LIN {X 79.235,Y 62.492,Z 71.887,A 180.000,B 0.000,C 180.000} C_DIS
LIN {X 78.583,Y 62.492,Z 72.273,A 180.000,B 0.000,C 180.000} C_DIS
LIN {X 77.938,Y 62.492,Z 72.685,A 180.000,B 0.000,C 180.000} C_DIS
LIN {X 77.253,Y 62.492,Z 73.150,A 180.000,B 0.000,C 180.000} C_DIS
LIN {X 76.356,Y 62.492,Z 73.799,A 180.000,B 0.000,C 180.000} C_DIS
LIN {X 75.526,Y 62.492,Z 74.437,A 180.000,B 0.000,C 180.000} C_DIS
LIN {X 74.385,Y 62.492,Z 75.346,A 180.000,B 0.000,C 180.000} C_DIS
LIN {X 71.167,Y 62.492,Z 77.984,A 180.000,B 0.000,C 180.000} C_DIS
LIN {X 70.008,Y 62.492,Z 78.896,A 180.000,B 0.000,C 180.000} C_DIS
LIN {X 69.397,Y 62.492,Z 79.356,A 180.000,B 0.000,C 180.000} C_DIS
LIN {X 68.827,Y 62.492,Z 79.771,A 180.000,B 0.000,C 180.000} C_DIS
LIN {X 68.251,Y 62.492,Z 80.172,A 180.000,B 0.000,C 180.000} C_DIS
LIN {X 67.665,Y 62.492,Z 80.560,A 180.000,B 0.000,C 180.000} C_DIS
LIN {X 67.072,Y 62.492,Z 80.930,A 180.000,B 0.000,C 180.000} C_DIS
LIN {X 66.471,Y 62.492,Z 81.280,A 180.000,B 0.000,C 180.000} C_DIS
LIN {X 65.863,Y 62.492,Z 81.607,A 180.000,B 0.000,C 180.000} C_DIS
LIN {X 65.243,Y 62.492,Z 81.911,A 180.000,B 0.000,C 180.000} C_DIS
LIN {X 64.615,Y 62.492,Z 82.187,A 180.000,B 0.000,C 180.000} C_DIS
LIN {X 63.980,Y 62.492,Z 82.433,A 180.000,B 0.000,C 180.000} C_DIS
LIN {X 63.335,Y 62.492,Z 82.646,A 180.000,B 0.000,C 180.000} C_DIS
LIN {X 62.690,Y 62.492,Z 82.823,A 180.000,B 0.000,C 180.000} C_DIS
LIN {X 62.017,Y 62.492,Z 82.967,A 180.000,B 0.000,C 180.000} C_DIS
LIN {X 61.641,Y 62.492,Z 83.029,A 180.000,B 0.000,C 180.000} C_DIS
LIN {X 61.284,Y 62.492,Z 83.076,A 180.000,B 0.000,C 180.000} C_DIS
LIN {X 60.974,Y 62.492,Z 83.108,A 180.000,B 0.000,C 180.000} C_DIS
LIN {X 60.606,Y 62.492,Z 83.133,A 180.000,B 0.000,C 180.000} C_DIS
LIN {X 60.279,Y 62.492,Z 83.146,A 180.000,B 0.000,C 180.000} C_DIS
LIN {X 59.499,Y 62.492,Z 83.150,A 180.000,B 0.000,C 180.000} C_DIS
LIN {X 54.601,Y 62.492,Z 83.148,A 180.000,B 0.000,C 180.000} C_DIS
LIN {X 54.227,Y 62.492,Z 83.136,A 180.000,B 0.000,C 180.000} C_DIS
LIN {X 53.915,Y 62.492,Z 83.117,A 180.000,B 0.000,C 180.000} C_DIS
LIN {X 53.559,Y 62.492,Z 83.084,A 180.000,B 0.000,C 180.000} C_DIS
LIN {X 53.202,Y 62.492,Z 83.039,A 180.000,B 0.000,C 180.000} C_DIS
LIN {X 52.828,Y 62.492,Z 82.980,A 180.000,B 0.000,C 180.000} C_DIS
LIN {X 52.471,Y 62.492,Z 82.912,A 180.000,B 0.000,C 180.000} C_DIS
LIN {X 52.095,Y 62.492,Z 82.827,A 180.000,B 0.000,C 180.000} C_DIS
LIN {X 51.709,Y 62.492,Z 82.727,A 180.000,B 0.000,C 180.000} C_DIS
LIN {X 51.331,Y 62.492,Z 82.617,A 180.000,B 0.000,C 180.000} C_DIS
LIN {X 50.942,Y 62.492,Z 82.490,A 180.000,B 0.000,C 180.000} C_DIS
LIN {X 50.561,Y 62.492,Z 82.354,A 180.000,B 0.000,C 180.000} C_DIS
LIN {X 50.167,Y 62.492,Z 82.199,A 180.000,B 0.000,C 180.000} C_DIS
LIN {X 49.770,Y 62.492,Z 82.030,A 180.000,B 0.000,C 180.000} C_DIS
LIN {X 49.363,Y 62.492,Z 81.843,A 180.000,B 0.000,C 180.000} C_DIS
LIN {X 48.958,Y 62.492,Z 81.643,A 180.000,B 0.000,C 180.000} C_DIS
LIN {X 48.549,Y 62.492,Z 81.428,A 180.000,B 0.000,C 180.000} C_DIS
LIN {X 48.135,Y 62.492,Z 81.196,A 180.000,B 0.000,C 180.000} C_DIS
LIN {X 47.721,Y 62.492,Z 80.950,A 180.000,B 0.000,C 180.000} C_DIS
LIN {X 47.296,Y 62.492,Z 80.683,A 180.000,B 0.000,C 180.000} C_DIS
LIN {X 46.964,Y 62.492,Z 80.467,A 180.000,B 0.000,C 180.000} C_DIS
LIN {X 46.964,Y 62.492,Z 62.000,A 180.000,B 0.000,C 180.000} C_DIS
LIN {X 23.973,Y 62.492,Z 62.000,A 180.000,B 0.000,C 180.000} C_DIS
LIN {X 23.973,Y 62.492,Z 57.000,A 180.000,B 0.000,C 180.000} C_DIS
LIN {X 4.022,Y 62.492,Z 57.000,A 180.000,B 0.000,C 180.000} C_DIS
LIN {X 4.022,Y 62.492,Z 52.000,A 180.000,B 0.000,C 180.000} C_DIS
LIN {X 2.500,Y 62.492,Z 52.000,A 180.000,B 0.000,C 180.000} C_DIS
LIN {X 2.500,Y 62.492,Z 45.000,A 180.000,B 0.000,C 180.000} C_DIS
LIN {X -0.010,Y 62.492,Z 45.000,A 180.000,B 0.000,C 180.000} C_DIS
; Link Move Starts
LIN {X -0.120,Y 62.492,Z 45.026,A 180.000,B 0.000,C 180.000} C_DIS
LIN {X -0.230,Y 62.492,Z 45.051,A 180.000,B 0.000,C 180.000} C_DIS
LIN {X -0.771,Y 62.804,Z 45.051,A 180.000,B 0.000,C 180.000} C_DIS
LIN {X -0.771,Y 63.429,Z 45.051,A 180.000,B 0.000,C 180.000} C_DIS
LIN {X -0.230,Y 63.742,Z 45.051,A 180.000,B 0.000,C 180.000} C_DIS
LIN {X -0.120,Y 63.742,Z 45.026,A 180.000,B 0.000,C 180.000} C_DIS
LIN {X -0.010,Y 63.742,Z 45.000,A 180.000,B 0.000,C 180.000} C_DIS
; Cutting Move Starts
LIN {X 2.500,Y 63.742,Z 45.000,A 180.000,B 0.000,C 180.000} C_DIS
LIN {X 2.500,Y 63.742,Z 52.000,A 180.000,B 0.000,C 180.000} C_DIS
LIN {X 3.774,Y 63.742,Z 52.000,A 180.000,B 0.000,C 180.000} C_DIS
LIN {X 3.775,Y 63.742,Z 57.000,A 180.000,B 0.000,C 180.000} C_DIS
LIN {X 22.723,Y 63.742,Z 57.000,A 180.000,B 0.000,C 180.000} C_DIS
LIN {X 22.723,Y 63.742,Z 62.000,A 180.000,B 0.000,C 180.000} C_DIS
LIN {X 47.384,Y 63.742,Z 62.000,A 180.000,B 0.000,C 180.000} C_DIS
LIN {X 47.386,Y 63.742,Z 80.467,A 180.000,B 0.000,C 180.000} C_DIS
LIN {X 47.722,Y 63.742,Z 80.686,A 180.000,B 0.000,C 180.000} C_DIS
LIN {X 48.142,Y 63.742,Z 80.950,A 180.000,B 0.000,C 180.000} C_DIS
LIN {X 48.557,Y 63.742,Z 81.195,A 180.000,B 0.000,C 180.000} C_DIS
LIN {X 48.971,Y 63.742,Z 81.427,A 180.000,B 0.000,C 180.000} C_DIS
LIN {X 49.380,Y 63.742,Z 81.643,A 180.000,B 0.000,C 180.000} C_DIS
LIN {X 49.785,Y 63.742,Z 81.843,A 180.000,B 0.000,C 180.000} C_DIS
LIN {X 50.192,Y 63.742,Z 82.030,A 180.000,B 0.000,C 180.000} C_DIS
LIN {X 50.588,Y 63.742,Z 82.199,A 180.000,B 0.000,C 180.000} C_DIS
LIN {X 50.974,Y 63.742,Z 82.350,A 180.000,B 0.000,C 180.000} C_DIS
LIN {X 51.364,Y 63.742,Z 82.490,A 180.000,B 0.000,C 180.000} C_DIS
LIN {X 51.752,Y 63.742,Z 82.617,A 180.000,B 0.000,C 180.000} C_DIS
LIN {X 52.130,Y 63.742,Z 82.727,A 180.000,B 0.000,C 180.000} C_DIS
LIN {X 52.516,Y 63.742,Z 82.827,A 180.000,B 0.000,C 180.000} C_DIS
LIN {X 52.892,Y 63.742,Z 82.912,A 180.000,B 0.000,C 180.000} C_DIS
LIN {X 53.250,Y 63.742,Z 82.980,A 180.000,B 0.000,C 180.000} C_DIS
LIN {X 53.623,Y 63.742,Z 83.039,A 180.000,B 0.000,C 180.000} C_DIS
LIN {X 53.981,Y 63.742,Z 83.084,A 180.000,B 0.000,C 180.000} C_DIS
LIN {X 54.336,Y 63.742,Z 83.117,A 180.000,B 0.000,C 180.000} C_DIS
LIN {X 54.649,Y 63.742,Z 83.136,A 180.000,B 0.000,C 180.000} C_DIS
LIN {X 55.023,Y 63.742,Z 83.148,A 180.000,B 0.000,C 180.000} C_DIS
LIN {X 59.920,Y 63.742,Z 83.150,A 180.000,B 0.000,C 180.000} C_DIS
LIN {X 60.700,Y 63.742,Z 83.146,A 180.000,B 0.000,C 180.000} C_DIS
LIN {X 61.027,Y 63.742,Z 83.134,A 180.000,B 0.000,C 180.000} C_DIS
LIN {X 61.394,Y 63.742,Z 83.108,A 180.000,B 0.000,C 180.000} C_DIS
LIN {X 61.705,Y 63.742,Z 83.076,A 180.000,B 0.000,C 180.000} C_DIS
LIN {X 62.062,Y 63.742,Z 83.029,A 180.000,B 0.000,C 180.000} C_DIS
LIN {X 62.438,Y 63.742,Z 82.967,A 180.000,B 0.000,C 180.000} C_DIS
LIN {X 63.111,Y 63.742,Z 82.823,A 180.000,B 0.000,C 180.000} C_DIS
LIN {X 63.766,Y 63.742,Z 82.643,A 180.000,B 0.000,C 180.000} C_DIS
LIN {X 64.410,Y 63.742,Z 82.430,A 180.000,B 0.000,C 180.000} C_DIS
LIN {X 65.044,Y 63.742,Z 82.185,A 180.000,B 0.000,C 180.000} C_DIS
LIN {X 65.664,Y 63.742,Z 81.912,A 180.000,B 0.000,C 180.000} C_DIS
LIN {X 66.284,Y 63.742,Z 81.608,A 180.000,B 0.000,C 180.000} C_DIS
LIN {X 66.891,Y 63.742,Z 81.281,A 180.000,B 0.000,C 180.000} C_DIS
LIN {X 67.493,Y 63.742,Z 80.930,A 180.000,B 0.000,C 180.000} C_DIS
LIN {X 68.086,Y 63.742,Z 80.560,A 180.000,B 0.000,C 180.000} C_DIS
LIN {X 68.672,Y 63.742,Z 80.172,A 180.000,B 0.000,C 180.000} C_DIS
LIN {X 69.248,Y 63.742,Z 79.771,A 180.000,B 0.000,C 180.000} C_DIS
LIN {X 69.818,Y 63.742,Z 79.357,A 180.000,B 0.000,C 180.000} C_DIS
LIN {X 70.434,Y 63.742,Z 78.893,A 180.000,B 0.000,C 180.000} C_DIS
LIN {X 71.592,Y 63.742,Z 77.980,A 180.000,B 0.000,C 180.000} C_DIS
LIN {X 74.778,Y 63.742,Z 75.369,A 180.000,B 0.000,C 180.000} C_DIS
LIN {X 76.394,Y 63.742,Z 74.080,A 180.000,B 0.000,C 180.000} C_DIS
LIN {X 77.534,Y 63.742,Z 73.194,A 180.000,B 0.000,C 180.000} C_DIS
LIN {X 78.214,Y 63.742,Z 72.684,A 180.000,B 0.000,C 180.000} C_DIS
LIN {X 78.784,Y 63.742,Z 72.272,A 180.000,B 0.000,C 180.000} C_DIS
LIN {X 79.325,Y 63.742,Z 71.899,A 180.000,B 0.000,C 180.000} C_DIS
LIN {X 79.847,Y 63.742,Z 71.559,A 180.000,B 0.000,C 180.000} C_DIS
LIN {X 80.351,Y 63.742,Z 71.251,A 180.000,B 0.000,C 180.000} C_DIS
LIN {X 80.842,Y 63.742,Z 70.974,A 180.000,B 0.000,C 180.000} C_DIS
LIN {X 81.321,Y 63.742,Z 70.730,A 180.000,B 0.000,C 180.000} C_DIS
LIN {X 81.779,Y 63.742,Z 70.521,A 180.000,B 0.000,C 180.000} C_DIS
LIN {X 82.174,Y 63.742,Z 70.367,A 180.000,B 0.000,C 180.000} C_DIS
LIN {X 82.462,Y 63.742,Z 70.265,A 180.000,B 0.000,C 180.000} C_DIS
LIN {X 82.842,Y 63.742,Z 70.159,A 180.000,B 0.000,C 180.000} C_DIS
LIN {X 83.153,Y 63.742,Z 70.096,A 180.000,B 0.000,C 180.000} C_DIS
LIN {X 83.373,Y 63.742,Z 70.085,A 180.000,B 0.000,C 180.000} C_DIS
LIN {X 83.458,Y 63.742,Z 70.072,A 180.000,B 0.000,C 180.000} C_DIS
LIN {X 83.461,Y 63.742,Z 62.000,A 180.000,B 0.000,C 180.000} C_DIS
LIN {X 132.277,Y 63.742,Z 62.000,A 180.000,B 0.000,C 180.000} C_DIS
LIN {X 132.277,Y 63.742,Z 57.000,A 180.000,B 0.000,C 180.000} C_DIS
LIN {X 151.225,Y 63.742,Z 57.000,A 180.000,B 0.000,C 180.000} C_DIS
LIN {X 151.225,Y 63.742,Z 52.000,A 180.000,B 0.000,C 180.000} C_DIS
LIN {X 152.500,Y 63.742,Z 52.000,A 180.000,B 0.000,C 180.000} C_DIS
LIN {X 152.500,Y 63.742,Z 45.000,A 180.000,B 0.000,C 180.000} C_DIS
LIN {X 155.010,Y 63.742,Z 45.000,A 180.000,B 0.000,C 180.000} C_DIS
; Link Move Starts
LIN {X 155.120,Y 63.742,Z 45.026,A 180.000,B 0.000,C 180.000} C_DIS
LIN {X 155.230,Y 63.742,Z 45.051,A 180.000,B 0.000,C 180.000} C_DIS
LIN {X 155.771,Y 64.054,Z 45.051,A 180.000,B 0.000,C 180.000} C_DIS
LIN {X 155.771,Y 64.679,Z 45.051,A 180.000,B 0.000,C 180.000} C_DIS
LIN {X 155.230,Y 64.991,Z 45.051,A 180.000,B 0.000,C 180.000} C_DIS
LIN {X 155.120,Y 64.991,Z 45.026,A 180.000,B 0.000,C 180.000} C_DIS
LIN {X 155.010,Y 64.991,Z 45.000,A 180.000,B 0.000,C 180.000} C_DIS
; Cutting Move Starts
LIN {X 152.500,Y 64.991,Z 45.000,A 180.000,B 0.000,C 180.000} C_DIS
LIN {X 152.500,Y 64.991,Z 52.000,A 180.000,B 0.000,C 180.000} C_DIS
LIN {X 151.447,Y 64.991,Z 52.000,A 180.000,B 0.000,C 180.000} C_DIS
LIN {X 151.444,Y 64.991,Z 57.000,A 180.000,B 0.000,C 180.000} C_DIS
LIN {X 133.527,Y 64.991,Z 57.000,A 180.000,B 0.000,C 180.000} C_DIS
LIN {X 133.525,Y 64.991,Z 62.000,A 180.000,B 0.000,C 180.000} C_DIS
LIN {X 79.755,Y 64.991,Z 62.000,A 180.000,B 0.000,C 180.000} C_DIS
LIN {X 79.752,Y 64.991,Z 70.826,A 180.000,B 0.000,C 180.000} C_DIS
LIN {X 79.714,Y 64.991,Z 70.913,A 180.000,B 0.000,C 180.000} C_DIS
LIN {X 79.604,Y 64.991,Z 71.063,A 180.000,B 0.000,C 180.000} C_DIS
LIN {X 79.296,Y 64.991,Z 71.377,A 180.000,B 0.000,C 180.000} C_DIS
LIN {X 78.473,Y 64.991,Z 72.127,A 180.000,B 0.000,C 180.000} C_DIS
LIN {X 77.133,Y 64.991,Z 73.359,A 180.000,B 0.000,C 180.000} C_DIS
LIN {X 75.322,Y 64.991,Z 75.057,A 180.000,B 0.000,C 180.000} C_DIS
LIN {X 74.334,Y 64.991,Z 75.972,A 180.000,B 0.000,C 180.000} C_DIS
LIN {X 73.331,Y 64.991,Z 76.866,A 180.000,B 0.000,C 180.000} C_DIS
LIN {X 72.319,Y 64.991,Z 77.730,A 180.000,B 0.000,C 180.000} C_DIS
LIN {X 71.861,Y 64.991,Z 78.101,A 180.000,B 0.000,C 180.000} C_DIS
LIN {X 70.854,Y 64.991,Z 78.894,A 180.000,B 0.000,C 180.000} C_DIS
LIN {X 70.239,Y 64.991,Z 79.358,A 180.000,B 0.000,C 180.000} C_DIS
LIN {X 69.669,Y 64.991,Z 79.772,A 180.000,B 0.000,C 180.000} C_DIS
LIN {X 69.093,Y 64.991,Z 80.173,A 180.000,B 0.000,C 180.000} C_DIS
LIN {X 68.507,Y 64.991,Z 80.561,A 180.000,B 0.000,C 180.000} C_DIS
LIN {X 67.914,Y 64.991,Z 80.931,A 180.000,B 0.000,C 180.000} C_DIS
LIN {X 67.312,Y 64.991,Z 81.281,A 180.000,B 0.000,C 180.000} C_DIS
LIN {X 66.705,Y 64.991,Z 81.608,A 180.000,B 0.000,C 180.000} C_DIS
LIN {X 66.084,Y 64.991,Z 81.912,A 180.000,B 0.000,C 180.000} C_DIS
LIN {X 65.464,Y 64.991,Z 82.185,A 180.000,B 0.000,C 180.000} C_DIS
LIN {X 64.831,Y 64.991,Z 82.430,A 180.000,B 0.000,C 180.000} C_DIS
LIN {X 64.187,Y 64.991,Z 82.643,A 180.000,B 0.000,C 180.000} C_DIS
LIN {X 63.532,Y 64.991,Z 82.823,A 180.000,B 0.000,C 180.000} C_DIS
LIN {X 62.858,Y 64.991,Z 82.967,A 180.000,B 0.000,C 180.000} C_DIS
LIN {X 62.483,Y 64.991,Z 83.029,A 180.000,B 0.000,C 180.000} C_DIS
LIN {X 62.153,Y 64.991,Z 83.073,A 180.000,B 0.000,C 180.000} C_DIS
LIN {X 61.815,Y 64.991,Z 83.108,A 180.000,B 0.000,C 180.000} C_DIS
LIN {X 61.447,Y 64.991,Z 83.134,A 180.000,B 0.000,C 180.000} C_DIS
LIN {X 61.121,Y 64.991,Z 83.146,A 180.000,B 0.000,C 180.000} C_DIS
LIN {X 60.342,Y 64.991,Z 83.150,A 180.000,B 0.000,C 180.000} C_DIS
LIN {X 55.445,Y 64.991,Z 83.148,A 180.000,B 0.000,C 180.000} C_DIS
LIN {X 55.111,Y 64.991,Z 83.138,A 180.000,B 0.000,C 180.000} C_DIS
LIN {X 54.764,Y 64.991,Z 83.117,A 180.000,B 0.000,C 180.000} C_DIS
LIN {X 54.409,Y 64.991,Z 83.085,A 180.000,B 0.000,C 180.000} C_DIS
LIN {X 54.051,Y 64.991,Z 83.040,A 180.000,B 0.000,C 180.000} C_DIS
LIN {X 53.674,Y 64.991,Z 82.980,A 180.000,B 0.000,C 180.000} C_DIS
LIN {X 53.314,Y 64.991,Z 82.912,A 180.000,B 0.000,C 180.000} C_DIS
LIN {X 52.938,Y 64.991,Z 82.827,A 180.000,B 0.000,C 180.000} C_DIS
LIN {X 52.552,Y 64.991,Z 82.727,A 180.000,B 0.000,C 180.000} C_DIS
LIN {X 52.174,Y 64.991,Z 82.617,A 180.000,B 0.000,C 180.000} C_DIS
LIN {X 51.786,Y 64.991,Z 82.491,A 180.000,B 0.000,C 180.000} C_DIS
LIN {X 51.404,Y 64.991,Z 82.354,A 180.000,B 0.000,C 180.000} C_DIS
LIN {X 51.010,Y 64.991,Z 82.199,A 180.000,B 0.000,C 180.000} C_DIS
LIN {X 50.613,Y 64.991,Z 82.030,A 180.000,B 0.000,C 180.000} C_DIS
LIN {X 50.206,Y 64.991,Z 81.843,A 180.000,B 0.000,C 180.000} C_DIS
LIN {X 49.802,Y 64.991,Z 81.643,A 180.000,B 0.000,C 180.000} C_DIS
LIN {X 49.393,Y 64.991,Z 81.428,A 180.000,B 0.000,C 180.000} C_DIS
LIN {X 48.979,Y 64.991,Z 81.196,A 180.000,B 0.000,C 180.000} C_DIS
LIN {X 48.564,Y 64.991,Z 80.950,A 180.000,B 0.000,C 180.000} C_DIS
LIN {X 48.139,Y 64.991,Z 80.683,A 180.000,B 0.000,C 180.000} C_DIS
LIN {X 47.807,Y 64.991,Z 80.467,A 180.000,B 0.000,C 180.000} C_DIS
LIN {X 47.807,Y 64.991,Z 62.000,A 180.000,B 0.000,C 180.000} C_DIS
LIN {X 21.473,Y 64.991,Z 62.000,A 180.000,B 0.000,C 180.000} C_DIS
LIN {X 21.473,Y 64.991,Z 57.000,A 180.000,B 0.000,C 180.000} C_DIS
LIN {X 3.553,Y 64.991,Z 57.000,A 180.000,B 0.000,C 180.000} C_DIS
LIN {X 3.551,Y 64.991,Z 52.000,A 180.000,B 0.000,C 180.000} C_DIS
LIN {X 2.500,Y 64.991,Z 52.000,A 180.000,B 0.000,C 180.000} C_DIS
LIN {X 2.500,Y 64.991,Z 45.000,A 180.000,B 0.000,C 180.000} C_DIS
LIN {X -0.010,Y 64.991,Z 45.000,A 180.000,B 0.000,C 180.000} C_DIS
; Link Move Starts
LIN {X -0.120,Y 64.991,Z 45.026,A 180.000,B 0.000,C 180.000} C_DIS
LIN {X -0.230,Y 64.991,Z 45.051,A 180.000,B 0.000,C 180.000} C_DIS
LIN {X -0.771,Y 65.304,Z 45.051,A 180.000,B 0.000,C 180.000} C_DIS
LIN {X -0.771,Y 65.929,Z 45.051,A 180.000,B 0.000,C 180.000} C_DIS
LIN {X -0.230,Y 66.241,Z 45.051,A 180.000,B 0.000,C 180.000} C_DIS
LIN {X -0.120,Y 66.241,Z 45.026,A 180.000,B 0.000,C 180.000} C_DIS
LIN {X -0.010,Y 66.241,Z 45.000,A 180.000,B 0.000,C 180.000} C_DIS
; Cutting Move Starts
LIN {X 2.496,Y 66.241,Z 45.000,A 180.000,B 0.000,C 180.000} C_DIS
LIN {X 2.500,Y 66.241,Z 52.000,A 180.000,B 0.000,C 180.000} C_DIS
LIN {X 3.355,Y 66.241,Z 52.000,A 180.000,B 0.000,C 180.000} C_DIS
LIN {X 3.355,Y 66.241,Z 57.000,A 180.000,B 0.000,C 180.000} C_DIS
LIN {X 20.223,Y 66.241,Z 57.000,A 180.000,B 0.000,C 180.000} C_DIS
LIN {X 20.223,Y 66.241,Z 62.000,A 180.000,B 0.000,C 180.000} C_DIS
LIN {X 48.229,Y 66.241,Z 62.000,A 180.000,B 0.000,C 180.000} C_DIS
LIN {X 48.229,Y 66.241,Z 80.467,A 180.000,B 0.000,C 180.000} C_DIS
LIN {X 48.566,Y 66.241,Z 80.686,A 180.000,B 0.000,C 180.000} C_DIS
LIN {X 48.986,Y 66.241,Z 80.949,A 180.000,B 0.000,C 180.000} C_DIS
LIN {X 49.400,Y 66.241,Z 81.195,A 180.000,B 0.000,C 180.000} C_DIS
LIN {X 49.814,Y 66.241,Z 81.427,A 180.000,B 0.000,C 180.000} C_DIS
LIN {X 50.223,Y 66.241,Z 81.643,A 180.000,B 0.000,C 180.000} C_DIS
LIN {X 50.628,Y 66.241,Z 81.843,A 180.000,B 0.000,C 180.000} C_DIS
LIN {X 51.035,Y 66.241,Z 82.030,A 180.000,B 0.000,C 180.000} C_DIS
LIN {X 51.432,Y 66.241,Z 82.199,A 180.000,B 0.000,C 180.000} C_DIS
LIN {X 51.826,Y 66.241,Z 82.354,A 180.000,B 0.000,C 180.000} C_DIS
LIN {X 52.207,Y 66.241,Z 82.491,A 180.000,B 0.000,C 180.000} C_DIS
LIN {X 52.596,Y 66.241,Z 82.617,A 180.000,B 0.000,C 180.000} C_DIS
LIN {X 52.974,Y 66.241,Z 82.727,A 180.000,B 0.000,C 180.000} C_DIS
LIN {X 53.360,Y 66.241,Z 82.827,A 180.000,B 0.000,C 180.000} C_DIS
LIN {X 53.736,Y 66.241,Z 82.912,A 180.000,B 0.000,C 180.000} C_DIS
LIN {X 54.096,Y 66.241,Z 82.980,A 180.000,B 0.000,C 180.000} C_DIS
LIN {X 54.473,Y 66.241,Z 83.040,A 180.000,B 0.000,C 180.000} C_DIS
LIN {X 54.830,Y 66.241,Z 83.085,A 180.000,B 0.000,C 180.000} C_DIS
LIN {X 55.186,Y 66.241,Z 83.118,A 180.000,B 0.000,C 180.000} C_DIS
LIN {X 55.533,Y 66.241,Z 83.138,A 180.000,B 0.000,C 180.000} C_DIS
LIN {X 55.866,Y 66.241,Z 83.148,A 180.000,B 0.000,C 180.000} C_DIS
LIN {X 60.763,Y 66.241,Z 83.150,A 180.000,B 0.000,C 180.000} C_DIS
LIN {X 61.540,Y 66.241,Z 83.146,A 180.000,B 0.000,C 180.000} C_DIS
LIN {X 61.867,Y 66.241,Z 83.134,A 180.000,B 0.000,C 180.000} C_DIS
LIN {X 62.235,Y 66.241,Z 83.108,A 180.000,B 0.000,C 180.000} C_DIS
LIN {X 62.572,Y 66.241,Z 83.073,A 180.000,B 0.000,C 180.000} C_DIS
LIN {X 62.902,Y 66.241,Z 83.029,A 180.000,B 0.000,C 180.000} C_DIS
LIN {X 63.278,Y 66.241,Z 82.968,A 180.000,B 0.000,C 180.000} C_DIS
LIN {X 63.951,Y 66.241,Z 82.823,A 180.000,B 0.000,C 180.000} C_DIS
LIN {X 64.607,Y 66.241,Z 82.644,A 180.000,B 0.000,C 180.000} C_DIS
LIN {X 65.252,Y 66.241,Z 82.430,A 180.000,B 0.000,C 180.000} C_DIS
LIN {X 65.886,Y 66.241,Z 82.185,A 180.000,B 0.000,C 180.000} C_DIS
LIN {X 66.506,Y 66.241,Z 81.912,A 180.000,B 0.000,C 180.000} C_DIS
LIN {X 67.126,Y 66.241,Z 81.608,A 180.000,B 0.000,C 180.000} C_DIS
LIN {X 67.733,Y 66.241,Z 81.282,A 180.000,B 0.000,C 180.000} C_DIS
LIN {X 68.300,Y 66.241,Z 80.952,A 180.000,B 0.000,C 180.000} C_DIS
LIN {X 68.878,Y 66.241,Z 80.587,A 180.000,B 0.000,C 180.000} C_DIS
LIN {X 69.434,Y 66.241,Z 80.205,A 180.000,B 0.000,C 180.000} C_DIS
LIN {X 69.976,Y 66.241,Z 79.805,A 180.000,B 0.000,C 180.000} C_DIS
LIN {X 70.536,Y 66.241,Z 79.363,A 180.000,B 0.000,C 180.000} C_DIS
LIN {X 71.204,Y 66.241,Z 78.797,A 180.000,B 0.000,C 180.000} C_DIS
LIN {X 72.107,Y 66.241,Z 77.965,A 180.000,B 0.000,C 180.000} C_DIS
LIN {X 72.821,Y 66.241,Z 77.253,A 180.000,B 0.000,C 180.000} C_DIS
LIN {X 73.563,Y 66.241,Z 76.474,A 180.000,B 0.000,C 180.000} C_DIS
LIN {X 74.250,Y 66.241,Z 75.709,A 180.000,B 0.000,C 180.000} C_DIS
LIN {X 74.780,Y 66.241,Z 75.079,A 180.000,B 0.000,C 180.000} C_DIS
LIN {X 75.196,Y 66.241,Z 74.560,A 180.000,B 0.000,C 180.000} C_DIS
LIN {X 75.567,Y 66.241,Z 74.047,A 180.000,B 0.000,C 180.000} C_DIS
LIN {X 75.795,Y 66.241,Z 73.692,A 180.000,B 0.000,C 180.000} C_DIS
LIN {X 75.931,Y 66.241,Z 73.439,A 180.000,B 0.000,C 180.000} C_DIS
LIN {X 76.016,Y 66.241,Z 73.226,A 180.000,B 0.000,C 180.000} C_DIS
LIN {X 76.048,Y 66.241,Z 73.082,A 180.000,B 0.000,C 180.000} C_DIS
LIN {X 76.050,Y 66.241,Z 62.000,A 180.000,B 0.000,C 180.000} C_DIS
LIN {X 134.777,Y 66.241,Z 62.000,A 180.000,B 0.000,C 180.000} C_DIS
LIN {X 134.777,Y 66.241,Z 57.000,A 180.000,B 0.000,C 180.000} C_DIS
LIN {X 151.643,Y 66.241,Z 57.000,A 180.000,B 0.000,C 180.000} C_DIS
LIN {X 151.645,Y 66.241,Z 52.000,A 180.000,B 0.000,C 180.000} C_DIS
LIN {X 152.500,Y 66.241,Z 52.000,A 180.000,B 0.000,C 180.000} C_DIS
LIN {X 152.500,Y 66.241,Z 45.000,A 180.000,B 0.000,C 180.000} C_DIS
LIN {X 155.010,Y 66.241,Z 45.000,A 180.000,B 0.000,C 180.000} C_DIS
; Link Move Starts
LIN {X 155.120,Y 66.241,Z 45.026,A 180.000,B 0.000,C 180.000} C_DIS
LIN {X 155.230,Y 66.241,Z 45.051,A 180.000,B 0.000,C 180.000} C_DIS
LIN {X 155.771,Y 66.554,Z 45.051,A 180.000,B 0.000,C 180.000} C_DIS
LIN {X 155.771,Y 67.179,Z 45.051,A 180.000,B 0.000,C 180.000} C_DIS
LIN {X 155.230,Y 67.491,Z 45.051,A 180.000,B 0.000,C 180.000} C_DIS
LIN {X 155.120,Y 67.491,Z 45.026,A 180.000,B 0.000,C 180.000} C_DIS
LIN {X 155.010,Y 67.491,Z 45.000,A 180.000,B 0.000,C 180.000} C_DIS
; Cutting Move Starts
LIN {X 152.500,Y 67.491,Z 45.000,A 180.000,B 0.000,C 180.000} C_DIS
LIN {X 152.500,Y 67.491,Z 52.000,A 180.000,B 0.000,C 180.000} C_DIS
LIN {X 151.825,Y 67.491,Z 52.000,A 180.000,B 0.000,C 180.000} C_DIS
LIN {X 151.825,Y 67.491,Z 57.000,A 180.000,B 0.000,C 180.000} C_DIS
LIN {X 136.027,Y 67.491,Z 57.000,A 180.000,B 0.000,C 180.000} C_DIS
LIN {X 136.027,Y 67.491,Z 62.000,A 180.000,B 0.000,C 180.000} C_DIS
LIN {X 72.345,Y 67.491,Z 62.000,A 180.000,B 0.000,C 180.000} C_DIS
LIN {X 72.341,Y 67.491,Z 76.312,A 180.000,B 0.000,C 180.000} C_DIS
LIN {X 72.307,Y 67.491,Z 76.482,A 180.000,B 0.000,C 180.000} C_DIS
LIN {X 72.222,Y 67.491,Z 76.719,A 180.000,B 0.000,C 180.000} C_DIS
LIN {X 72.072,Y 67.491,Z 77.028,A 180.000,B 0.000,C 180.000} C_DIS
LIN {X 71.857,Y 67.491,Z 77.390,A 180.000,B 0.000,C 180.000} C_DIS
LIN {X 71.559,Y 67.491,Z 77.830,A 180.000,B 0.000,C 180.000} C_DIS
LIN {X 71.235,Y 67.491,Z 78.249,A 180.000,B 0.000,C 180.000} C_DIS
LIN {X 70.751,Y 67.491,Z 78.822,A 180.000,B 0.000,C 180.000} C_DIS
LIN {X 70.256,Y 67.491,Z 79.345,A 180.000,B 0.000,C 180.000} C_DIS
LIN {X 69.786,Y 67.491,Z 79.800,A 180.000,B 0.000,C 180.000} C_DIS
LIN {X 69.333,Y 67.491,Z 80.203,A 180.000,B 0.000,C 180.000} C_DIS
LIN {X 68.864,Y 67.491,Z 80.587,A 180.000,B 0.000,C 180.000} C_DIS
LIN {X 68.375,Y 67.491,Z 80.955,A 180.000,B 0.000,C 180.000} C_DIS
LIN {X 67.865,Y 67.491,Z 81.301,A 180.000,B 0.000,C 180.000} C_DIS
LIN {X 67.336,Y 67.491,Z 81.626,A 180.000,B 0.000,C 180.000} C_DIS
LIN {X 66.786,Y 67.491,Z 81.925,A 180.000,B 0.000,C 180.000} C_DIS
LIN {X 66.211,Y 67.491,Z 82.199,A 180.000,B 0.000,C 180.000} C_DIS
LIN {X 65.615,Y 67.491,Z 82.441,A 180.000,B 0.000,C 180.000} C_DIS
LIN {X 64.994,Y 67.491,Z 82.652,A 180.000,B 0.000,C 180.000} C_DIS
LIN {X 64.375,Y 67.491,Z 82.823,A 180.000,B 0.000,C 180.000} C_DIS
LIN {X 63.702,Y 67.491,Z 82.967,A 180.000,B 0.000,C 180.000} C_DIS
LIN {X 63.327,Y 67.491,Z 83.029,A 180.000,B 0.000,C 180.000} C_DIS
LIN {X 62.969,Y 67.491,Z 83.076,A 180.000,B 0.000,C 180.000} C_DIS
LIN {X 62.659,Y 67.491,Z 83.108,A 180.000,B 0.000,C 180.000} C_DIS
LIN {X 62.287,Y 67.491,Z 83.134,A 180.000,B 0.000,C 180.000} C_DIS
LIN {X 62.026,Y 67.491,Z 83.145,A 180.000,B 0.000,C 180.000} C_DIS
LIN {X 60.940,Y 67.491,Z 83.150,A 180.000,B 0.000,C 180.000} C_DIS
LIN {X 56.288,Y 67.491,Z 83.148,A 180.000,B 0.000,C 180.000} C_DIS
LIN {X 55.954,Y 67.491,Z 83.138,A 180.000,B 0.000,C 180.000} C_DIS
LIN {X 55.607,Y 67.491,Z 83.117,A 180.000,B 0.000,C 180.000} C_DIS
LIN {X 55.251,Y 67.491,Z 83.085,A 180.000,B 0.000,C 180.000} C_DIS
LIN {X 54.894,Y 67.491,Z 83.040,A 180.000,B 0.000,C 180.000} C_DIS
LIN {X 54.517,Y 67.491,Z 82.980,A 180.000,B 0.000,C 180.000} C_DIS
LIN {X 54.157,Y 67.491,Z 82.912,A 180.000,B 0.000,C 180.000} C_DIS
LIN {X 53.781,Y 67.491,Z 82.827,A 180.000,B 0.000,C 180.000} C_DIS
LIN {X 53.395,Y 67.491,Z 82.727,A 180.000,B 0.000,C 180.000} C_DIS
LIN {X 53.018,Y 67.491,Z 82.617,A 180.000,B 0.000,C 180.000} C_DIS
LIN {X 52.630,Y 67.491,Z 82.491,A 180.000,B 0.000,C 180.000} C_DIS
LIN {X 52.240,Y 67.491,Z 82.351,A 180.000,B 0.000,C 180.000} C_DIS
LIN {X 51.847,Y 67.491,Z 82.196,A 180.000,B 0.000,C 180.000} C_DIS
LIN {X 51.450,Y 67.491,Z 82.027,A 180.000,B 0.000,C 180.000} C_DIS
LIN {X 51.050,Y 67.491,Z 81.843,A 180.000,B 0.000,C 180.000} C_DIS
LIN {X 50.645,Y 67.491,Z 81.643,A 180.000,B 0.000,C 180.000} C_DIS
LIN {X 50.236,Y 67.491,Z 81.428,A 180.000,B 0.000,C 180.000} C_DIS
LIN {X 49.822,Y 67.491,Z 81.196,A 180.000,B 0.000,C 180.000} C_DIS
LIN {X 49.408,Y 67.491,Z 80.950,A 180.000,B 0.000,C 180.000} C_DIS
LIN {X 48.982,Y 67.491,Z 80.683,A 180.000,B 0.000,C 180.000} C_DIS
LIN {X 48.651,Y 67.491,Z 80.467,A 180.000,B 0.000,C 180.000} C_DIS
LIN {X 48.649,Y 67.491,Z 62.000,A 180.000,B 0.000,C 180.000} C_DIS
LIN {X 18.973,Y 67.491,Z 62.000,A 180.000,B 0.000,C 180.000} C_DIS
LIN {X 18.973,Y 67.491,Z 57.000,A 180.000,B 0.000,C 180.000} C_DIS
LIN {X 3.175,Y 67.491,Z 57.000,A 180.000,B 0.000,C 180.000} C_DIS
LIN {X 3.175,Y 67.491,Z 52.000,A 180.000,B 0.000,C 180.000} C_DIS
LIN {X 2.500,Y 67.491,Z 52.000,A 180.000,B 0.000,C 180.000} C_DIS
LIN {X 2.500,Y 67.491,Z 45.000,A 180.000,B 0.000,C 180.000} C_DIS
LIN {X -0.010,Y 67.491,Z 45.000,A 180.000,B 0.000,C 180.000} C_DIS
; Link Move Starts
LIN {X -0.120,Y 67.491,Z 45.026,A 180.000,B 0.000,C 180.000} C_DIS
LIN {X -0.230,Y 67.491,Z 45.051,A 180.000,B 0.000,C 180.000} C_DIS
LIN {X -0.771,Y 67.804,Z 45.051,A 180.000,B 0.000,C 180.000} C_DIS
LIN {X -0.771,Y 68.429,Z 45.051,A 180.000,B 0.000,C 180.000} C_DIS
LIN {X -0.230,Y 68.741,Z 45.051,A 180.000,B 0.000,C 180.000} C_DIS
LIN {X -0.120,Y 68.741,Z 45.026,A 180.000,B 0.000,C 180.000} C_DIS
LIN {X -0.010,Y 68.741,Z 45.000,A 180.000,B 0.000,C 180.000} C_DIS
; Cutting Move Starts
LIN {X 2.500,Y 68.741,Z 45.000,A 180.000,B 0.000,C 180.000} C_DIS
LIN {X 2.500,Y 68.741,Z 52.000,A 180.000,B 0.000,C 180.000} C_DIS
LIN {X 3.013,Y 68.741,Z 52.000,A 180.000,B 0.000,C 180.000} C_DIS
LIN {X 3.013,Y 68.741,Z 57.000,A 180.000,B 0.000,C 180.000} C_DIS
LIN {X 17.723,Y 68.741,Z 57.000,A 180.000,B 0.000,C 180.000} C_DIS
LIN {X 17.723,Y 68.741,Z 62.000,A 180.000,B 0.000,C 180.000} C_DIS
LIN {X 49.071,Y 68.741,Z 62.000,A 180.000,B 0.000,C 180.000} C_DIS
LIN {X 49.072,Y 68.741,Z 80.467,A 180.000,B 0.000,C 180.000} C_DIS
LIN {X 49.404,Y 68.741,Z 80.683,A 180.000,B 0.000,C 180.000} C_DIS
LIN {X 49.829,Y 68.741,Z 80.950,A 180.000,B 0.000,C 180.000} C_DIS
LIN {X 50.244,Y 68.741,Z 81.196,A 180.000,B 0.000,C 180.000} C_DIS
LIN {X 50.658,Y 68.741,Z 81.428,A 180.000,B 0.000,C 180.000} C_DIS
LIN {X 51.067,Y 68.741,Z 81.643,A 180.000,B 0.000,C 180.000} C_DIS
LIN {X 51.472,Y 68.741,Z 81.843,A 180.000,B 0.000,C 180.000} C_DIS
LIN {X 51.872,Y 68.741,Z 82.027,A 180.000,B 0.000,C 180.000} C_DIS
LIN {X 52.268,Y 68.741,Z 82.196,A 180.000,B 0.000,C 180.000} C_DIS
LIN {X 52.662,Y 68.741,Z 82.351,A 180.000,B 0.000,C 180.000} C_DIS
LIN {X 53.051,Y 68.741,Z 82.491,A 180.000,B 0.000,C 180.000} C_DIS
LIN {X 53.440,Y 68.741,Z 82.617,A 180.000,B 0.000,C 180.000} C_DIS
LIN {X 53.817,Y 68.741,Z 82.727,A 180.000,B 0.000,C 180.000} C_DIS
LIN {X 54.203,Y 68.741,Z 82.827,A 180.000,B 0.000,C 180.000} C_DIS
LIN {X 54.579,Y 68.741,Z 82.912,A 180.000,B 0.000,C 180.000} C_DIS
LIN {X 54.939,Y 68.741,Z 82.980,A 180.000,B 0.000,C 180.000} C_DIS
LIN {X 55.316,Y 68.741,Z 83.040,A 180.000,B 0.000,C 180.000} C_DIS
LIN {X 55.673,Y 68.741,Z 83.085,A 180.000,B 0.000,C 180.000} C_DIS
LIN {X 56.029,Y 68.741,Z 83.117,A 180.000,B 0.000,C 180.000} C_DIS
LIN {X 56.376,Y 68.741,Z 83.138,A 180.000,B 0.000,C 180.000} C_DIS
LIN {X 56.676,Y 68.741,Z 83.147,A 180.000,B 0.000,C 180.000} C_DIS
LIN {X 62.175,Y 68.741,Z 83.148,A 180.000,B 0.000,C 180.000} C_DIS
LIN {X 62.572,Y 68.741,Z 83.137,A 180.000,B 0.000,C 180.000} C_DIS
LIN {X 63.009,Y 68.741,Z 83.105,A 180.000,B 0.000,C 180.000} C_DIS
LIN {X 63.472,Y 68.741,Z 83.046,A 180.000,B 0.000,C 180.000} C_DIS
LIN {X 63.871,Y 68.741,Z 82.975,A 180.000,B 0.000,C 180.000} C_DIS
LIN {X 64.463,Y 68.741,Z 82.829,A 180.000,B 0.000,C 180.000} C_DIS
LIN {X 65.010,Y 68.741,Z 82.652,A 180.000,B 0.000,C 180.000} C_DIS
LIN {X 65.529,Y 68.741,Z 82.442,A 180.000,B 0.000,C 180.000} C_DIS
LIN {X 66.027,Y 68.741,Z 82.198,A 180.000,B 0.000,C 180.000} C_DIS
LIN {X 66.501,Y 68.741,Z 81.923,A 180.000,B 0.000,C 180.000} C_DIS
LIN {X 66.951,Y 68.741,Z 81.617,A 180.000,B 0.000,C 180.000} C_DIS
LIN {X 67.368,Y 68.741,Z 81.288,A 180.000,B 0.000,C 180.000} C_DIS
LIN {X 67.730,Y 68.741,Z 80.957,A 180.000,B 0.000,C 180.000} C_DIS
LIN {X 67.972,Y 68.741,Z 80.704,A 180.000,B 0.000,C 180.000} C_DIS
LIN {X 68.190,Y 68.741,Z 80.447,A 180.000,B 0.000,C 180.000} C_DIS
LIN {X 68.398,Y 68.741,Z 80.155,A 180.000,B 0.000,C 180.000} C_DIS
LIN {X 68.524,Y 68.741,Z 79.930,A 180.000,B 0.000,C 180.000} C_DIS
LIN {X 68.602,Y 68.741,Z 79.738,A 180.000,B 0.000,C 180.000} C_DIS
LIN {X 68.636,Y 68.741,Z 79.588,A 180.000,B 0.000,C 180.000} C_DIS
LIN {X 68.640,Y 68.741,Z 62.000,A 180.000,B 0.000,C 180.000} C_DIS
LIN {X 137.277,Y 68.741,Z 62.000,A 180.000,B 0.000,C 180.000} C_DIS
LIN {X 137.277,Y 68.741,Z 57.000,A 180.000,B 0.000,C 180.000} C_DIS
LIN {X 151.987,Y 68.741,Z 57.000,A 180.000,B 0.000,C 180.000} C_DIS
